C03648=1197.053,12.345,-44.404,-179.678,5.675,148.906
C03649=1197.057,12.095,-44.389,-179.681,5.675,148.907
C03650=1197.063,11.846,-44.375,-179.684,5.674,148.908
C03651=1197.069,11.596,-44.360,-179.686,5.674,148.908
C03652=1197.074,11.347,-44.346,-179.689,5.673,148.909
C03653=1197.079,11.097,-44.331,-179.691,5.672,148.910
C03654=1197.084,10.847,-44.317,-179.694,5.672,148.910
C03655=1197.088,10.598,-44.302,-179.697,5.671,148.911
C03656=1197.093,10.349,-44.288,-179.699,5.671,148.912
C03657=1197.099,10.100,-44.274,-179.702,5.670,148.912
C03658=1197.104,9.850,-44.260,-179.704,5.669,148.913
C03659=1197.109,9.600,-44.245,-179.707,5.669,148.914
C03660=1197.114,9.350,-44.231,-179.709,5.669,148.914
C03661=1197.119,9.101,-44.217,-179.712,5.668,148.915
C03662=1197.123,8.851,-44.203,-179.714,5.667,148.915
C03663=1197.129,8.602,-44.189,-179.717,5.667,148.916
C03664=1197.134,8.352,-44.174,-179.719,5.667,148.917
C03665=1197.139,8.103,-44.159,-179.721,5.666,148.917
C03666=1197.144,7.853,-44.145,-179.724,5.666,148.918
C03667=1197.149,7.604,-44.131,-179.726,5.665,148.919
C03668=1197.154,7.355,-44.117,-179.729,5.665,148.919
C03669=1197.159,7.105,-44.103,-179.732,5.664,148.920
C03670=1197.164,6.855,-44.088,-179.734,5.664,148.921
C03671=1197.169,6.606,-44.074,-179.737,5.663,148.921
C03672=1197.174,6.356,-44.060,-179.739,5.662,148.922
C03673=1197.179,6.107,-44.046,-179.742,5.662,148.922
C03674=1197.184,5.857,-44.032,-179.744,5.661,148.923
C03675=1197.189,5.607,-44.017,-179.747,5.661,148.924
C03676=1197.194,5.358,-44.003,-179.750,5.660,148.924
C03677=1197.200,5.109,-43.989,-179.751,5.660,148.925
C03678=1197.205,4.858,-43.976,-179.754,5.660,148.926
C03679=1197.209,4.609,-43.962,-179.757,5.659,148.926
C03680=1197.214,4.359,-43.948,-179.759,5.659,148.927
C03681=1197.220,4.110,-43.934,-179.762,5.658,148.928
C03682=1197.225,3.861,-43.919,-179.764,5.657,148.928
C03683=1197.230,3.611,-43.905,-179.767,5.657,148.929
C03684=1197.235,3.361,-43.891,-179.769,5.656,148.930
C03685=1197.241,3.092,-43.876,-179.772,5.656,148.930
C03686=1197.246,2.824,-43.861,-179.775,5.655,148.931
C03687=1197.251,2.554,-43.846,-179.777,5.655,148.932
C03688=1197.257,2.285,-43.831,-179.780,5.654,148.932
C03689=1197.262,2.035,-43.816,-179.783,5.654,148.933
C03690=1197.267,1.786,-43.802,-179.785,5.653,148.934
C03691=1197.272,1.536,-43.788,-179.788,5.653,148.934
C03692=1197.277,1.286,-43.775,-179.790,5.652,148.935
C03693=1197.282,1.037,-43.761,-179.793,5.652,148.935
C03694=1197.287,0.788,-43.747,-179.795,5.652,148.936
C03695=1197.292,0.538,-43.733,-179.797,5.651,148.937
C03696=1197.298,0.289,-43.719,-179.800,5.651,148.938
C03697=1197.303,0.039,-43.705,-179.802,5.650,148.938
C03698=1197.307,-0.211,-43.692,-179.805,5.650,148.939
C03699=1197.313,-0.460,-43.678,-179.808,5.649,148.939
C03700=1197.318,-0.710,-43.663,-179.810,5.649,148.940
C03701=1197.323,-0.959,-43.649,-179.813,5.648,148.941
C03702=1197.329,-1.209,-43.636,-179.815,5.647,148.941
C03703=1197.333,-1.458,-43.622,-179.817,5.648,148.942
C03704=1197.338,-1.708,-43.608,-179.820,5.647,148.943
C03705=1197.343,-1.957,-43.594,-179.822,5.647,148.943
C03706=1197.349,-2.207,-43.580,-179.825,5.646,148.944
C03707=1197.353,-2.457,-43.567,-179.827,5.645,148.944
C03708=1197.358,-2.706,-43.553,-179.830,5.645,148.945
C03709=1197.364,-2.956,-43.539,-179.833,5.644,148.946
C03710=1197.369,-3.206,-43.525,-179.835,5.644,148.947
C03711=1197.373,-3.454,-43.512,-179.837,5.644,148.947
C03712=1197.379,-3.705,-43.498,-179.840,5.644,148.948
C03713=1197.384,-3.954,-43.484,-179.842,5.643,148.948
C03714=1197.389,-4.204,-43.470,-179.845,5.642,148.949
C03715=1197.394,-4.454,-43.457,-179.847,5.642,148.950
C03716=1197.399,-4.703,-43.443,-179.850,5.641,148.950
C03717=1197.404,-4.952,-43.429,-179.853,5.641,148.951
C03718=1197.409,-5.203,-43.415,-179.855,5.640,148.952
C03719=1197.414,-5.451,-43.402,-179.857,5.640,148.952
C03720=1197.419,-5.701,-43.388,-179.860,5.640,148.953
C03721=1197.425,-5.951,-43.374,-179.862,5.639,148.954
C03722=1197.429,-6.200,-43.361,-179.865,5.639,148.954
C03723=1197.435,-6.450,-43.347,-179.867,5.638,148.955
C03724=1197.440,-6.699,-43.333,-179.870,5.638,148.955
C03725=1197.445,-6.949,-43.320,-179.872,5.637,148.956
C03726=1197.450,-7.198,-43.306,-179.874,5.637,148.957
C03727=1197.455,-7.448,-43.292,-179.877,5.637,148.958
C03728=1197.460,-7.698,-43.279,-179.880,5.636,148.958
C03729=1197.465,-7.947,-43.265,-179.882,5.636,148.959
C03730=1197.470,-8.197,-43.252,-179.885,5.635,148.959
C03731=1197.475,-8.446,-43.238,-179.887,5.635,148.960
C03732=1197.481,-8.696,-43.225,-179.890,5.634,148.961
C03733=1197.485,-8.945,-43.211,-179.892,5.634,148.961
C03734=1197.491,-9.196,-43.198,-179.894,5.634,148.962
C03735=1197.495,-9.444,-43.185,-179.897,5.633,148.963
C03736=1197.501,-9.695,-43.171,-179.899,5.633,148.963
C03737=1197.506,-9.944,-43.157,-179.902,5.632,148.964
C03738=1197.511,-10.194,-43.144,-179.905,5.632,148.965
C03739=1197.516,-10.443,-43.130,-179.907,5.631,148.965
C03740=1197.521,-10.693,-43.117,-179.909,5.631,148.966
C03741=1197.526,-10.942,-43.103,-179.912,5.631,148.967
C03742=1197.532,-11.192,-43.090,-179.914,5.630,148.967
C03743=1197.536,-11.442,-43.077,-179.917,5.630,148.968
C03744=1197.542,-11.691,-43.063,-179.920,5.629,148.969
C03745=1197.546,-11.941,-43.050,-179.922,5.628,148.969
C03746=1197.552,-12.190,-43.036,-179.924,5.629,148.970
C03747=1197.556,-12.440,-43.023,-179.927,5.628,148.970
C03748=1197.562,-12.690,-43.010,-179.929,5.628,148.971
C03749=1197.566,-12.939,-42.996,-179.932,5.627,148.972
C03750=1197.572,-13.189,-42.983,-179.934,5.626,148.972
C03751=1197.577,-13.438,-42.969,-179.937,5.626,148.973
C03752=1197.582,-13.688,-42.956,-179.939,5.626,148.974
C03753=1197.587,-13.938,-42.943,-179.941,5.626,148.974
C03754=1197.592,-14.187,-42.929,-179.944,5.625,148.975
C03755=1197.597,-14.437,-42.916,-179.947,5.625,148.976
C03756=1197.603,-14.686,-42.903,-179.949,5.624,148.976
C03757=1197.608,-14.935,-42.890,-179.952,5.623,148.977
C03758=1197.613,-15.185,-42.876,-179.954,5.624,148.978
C03759=1197.618,-15.435,-42.864,-179.956,5.623,148.978
C03760=1197.623,-15.685,-42.850,-179.959,5.623,148.979
C03761=1197.628,-15.934,-42.837,-179.961,5.622,148.980
C03762=1197.633,-16.184,-42.823,-179.964,5.622,148.980
C03763=1197.639,-16.433,-42.811,-179.966,5.622,148.981
C03764=1197.643,-16.683,-42.797,-179.969,5.621,148.982
C03765=1197.649,-16.932,-42.784,-179.971,5.621,148.982
C03766=1197.654,-17.182,-42.771,-179.974,5.620,148.983
C03767=1197.659,-17.432,-42.758,-179.976,5.620,148.983
C03768=1197.664,-17.681,-42.744,-179.979,5.619,148.984
C03769=1197.669,-17.931,-42.731,-179.981,5.619,148.985
C03770=1197.674,-18.180,-42.718,-179.983,5.619,148.986
C03771=1197.679,-18.430,-42.705,-179.986,5.619,148.986
C03772=1197.685,-18.680,-42.692,-179.989,5.618,148.987
C03773=1197.689,-18.929,-42.679,-179.991,5.617,148.987
C03774=1197.695,-19.179,-42.665,-179.993,5.618,148.988
C03775=1197.700,-19.428,-42.652,-179.996,5.617,148.989
C03776=1197.704,-19.678,-42.639,-179.998,5.617,148.989
C03777=1197.710,-19.928,-42.626,179.999,5.616,148.990
C03778=1197.715,-20.177,-42.614,179.997,5.615,148.991
C03779=1197.720,-20.427,-42.599,179.995,5.616,148.991
C03780=1197.725,-20.676,-42.587,179.992,5.615,148.992
C03781=1197.730,-20.926,-42.574,179.989,5.615,148.993
C03782=1197.736,-21.176,-42.561,179.987,5.614,148.993
C03783=1197.741,-21.425,-42.548,179.984,5.614,148.994
C03784=1197.746,-21.675,-42.535,179.983,5.614,148.995
C03785=1197.751,-21.925,-42.522,179.980,5.613,148.995
C03786=1197.756,-22.174,-42.509,179.977,5.613,148.996
C03787=1197.761,-22.424,-42.496,179.975,5.612,148.997
C03788=1197.766,-22.673,-42.482,179.972,5.612,148.997
C03789=1197.771,-22.943,-42.469,179.969,5.611,148.998
C03790=1197.778,-23.212,-42.455,179.967,5.612,148.999
C03791=1197.783,-23.482,-42.441,179.965,5.611,148.999
C03792=1197.789,-23.752,-42.427,179.962,5.611,149.000
C03793=1197.794,-24.001,-42.414,179.959,5.610,149.001
C03794=1197.799,-24.251,-42.402,179.957,5.610,149.002
C03795=1197.803,-24.501,-42.389,179.954,5.609,149.002
C03796=1197.809,-24.750,-42.375,179.952,5.609,149.003
C03797=1197.814,-25.000,-42.363,179.950,5.609,149.003
C03798=1197.819,-25.250,-42.350,179.947,5.608,149.004
C03799=1197.824,-25.499,-42.337,179.944,5.608,149.005
C03800=1197.830,-25.749,-42.324,179.942,5.607,149.005
C03801=1197.835,-25.998,-42.312,179.940,5.607,149.006
C03802=1197.839,-26.248,-42.299,179.937,5.607,149.007
C03803=1197.845,-26.497,-42.286,179.935,5.606,149.007
C03804=1197.850,-26.747,-42.273,179.932,5.606,149.008
C03805=1197.855,-26.997,-42.260,179.930,5.606,149.009
C03806=1197.860,-27.246,-42.247,179.928,5.605,149.009
C03807=1197.865,-27.496,-42.235,179.925,5.605,149.010
C03808=1197.870,-27.746,-42.222,179.923,5.605,149.011
C03809=1197.876,-27.995,-42.208,179.920,5.604,149.011
C03810=1197.881,-28.245,-42.196,179.918,5.604,149.012
C03811=1197.886,-28.495,-42.184,179.915,5.604,149.013
C03812=1197.891,-28.745,-42.171,179.913,5.603,149.013
C03813=1197.896,-28.994,-42.158,179.910,5.603,149.014
C03814=1197.901,-29.243,-42.146,179.908,5.603,149.015
C03815=1197.907,-29.493,-42.133,179.906,5.602,149.015
C03816=1197.911,-29.743,-42.120,179.903,5.602,149.016
C03817=1197.916,-29.992,-42.107,179.901,5.601,149.016
C03818=1197.922,-30.242,-42.094,179.899,5.602,149.017
C03819=1197.927,-30.491,-42.083,179.896,5.601,149.018
C03820=1197.931,-30.741,-42.070,179.893,5.601,149.019
C03821=1197.937,-30.991,-42.057,179.891,5.600,149.019
C03822=1197.942,-31.240,-42.044,179.889,5.600,149.020
C03823=1197.948,-31.490,-42.031,179.886,5.600,149.020
C03824=1197.953,-31.740,-42.019,179.884,5.599,149.021
C03825=1197.958,-31.990,-42.006,179.881,5.599,149.022
C03826=1197.963,-32.239,-41.994,179.879,5.599,149.022
C03827=1197.968,-32.488,-41.981,179.876,5.599,149.023
C03828=1197.973,-32.738,-41.968,179.874,5.598,149.024
C03829=1197.978,-32.988,-41.957,179.872,5.597,149.024
C03830=1197.983,-33.238,-41.944,179.869,5.598,149.025
C03831=1197.988,-33.487,-41.931,179.867,5.597,149.026
C03832=1197.994,-33.737,-41.918,179.864,5.597,149.026
C03833=1197.999,-33.986,-41.906,179.861,5.596,149.027
C03834=1198.004,-34.236,-41.893,179.860,5.596,149.028
C03835=1198.009,-34.486,-41.880,179.857,5.596,149.028
C03836=1198.014,-34.736,-41.869,179.855,5.595,149.029
C03837=1198.019,-34.985,-41.856,179.852,5.595,149.030
C03838=1198.025,-35.234,-41.843,179.850,5.595,149.030
C03839=1198.030,-35.484,-41.831,179.847,5.595,149.031
C03840=1198.035,-35.734,-41.819,179.845,5.594,149.032
C03841=1198.040,-35.984,-41.806,179.842,5.593,149.032
C03842=1198.045,-36.233,-41.793,179.840,5.594,149.033
C03843=1198.050,-36.483,-41.781,179.838,5.593,149.034
C03844=1198.055,-36.732,-41.769,179.835,5.593,149.034
C03845=1198.061,-36.982,-41.757,179.833,5.592,149.035
C03846=1198.066,-37.231,-41.744,179.831,5.592,149.036
C03847=1198.071,-37.481,-41.732,179.828,5.592,149.036
C03848=1198.076,-37.731,-41.720,179.825,5.591,149.037
C03849=1198.081,-37.981,-41.707,179.823,5.591,149.038
C03850=1198.086,-38.230,-41.694,179.821,5.591,149.038
C03851=1198.092,-38.480,-41.682,179.818,5.590,149.039
C03852=1198.097,-38.729,-41.670,179.816,5.590,149.040
C03853=1198.102,-38.979,-41.658,179.814,5.590,149.040
C03854=1198.107,-39.229,-41.645,179.811,5.590,149.041
C03855=1198.113,-39.479,-41.633,179.808,5.589,149.042
C03856=1198.118,-39.728,-41.621,179.806,5.589,149.042
C03857=1198.123,-39.977,-41.608,179.804,5.589,149.043
C03858=1198.128,-40.228,-41.596,179.801,5.589,149.043
C03859=1198.132,-40.477,-41.584,179.799,5.588,149.044
C03860=1198.138,-40.727,-41.572,179.797,5.588,149.045
C03861=1198.143,-40.976,-41.559,179.794,5.588,149.046
C03862=1198.148,-41.226,-41.548,179.792,5.587,149.046
C03863=1198.153,-41.475,-41.535,179.789,5.587,149.047
C03864=1198.159,-41.725,-41.523,179.787,5.587,149.047
C03865=1198.164,-41.975,-41.510,179.784,5.587,149.048
C03866=1198.169,-42.224,-41.499,179.782,5.586,149.049
C03867=1198.174,-42.474,-41.486,179.780,5.586,149.049
C03868=1198.180,-42.724,-41.474,179.777,5.586,149.050
C03869=1198.184,-42.973,-41.462,179.775,5.585,149.051
C03870=1198.190,-43.223,-41.450,179.772,5.585,149.051
C03871=1198.195,-43.473,-41.438,179.770,5.585,149.052
C03872=1198.200,-43.723,-41.425,179.767,5.585,149.053
C03873=1198.205,-43.973,-41.413,179.765,5.584,149.053
C03874=1198.210,-44.222,-41.401,179.763,5.584,149.054
C03875=1198.215,-44.472,-41.390,179.760,5.584,149.055
C03876=1198.220,-44.721,-41.377,179.758,5.583,149.055
C03877=1198.225,-44.971,-41.365,179.755,5.583,149.056
C03878=1198.231,-45.221,-41.353,179.754,5.583,149.057
C03879=1198.236,-45.470,-41.341,179.751,5.582,149.057
C03880=1198.241,-45.720,-41.329,179.748,5.582,149.058
C03881=1198.246,-45.969,-41.317,179.746,5.582,149.059
C03882=1198.251,-46.219,-41.305,179.743,5.582,149.059
C03883=1198.257,-46.469,-41.293,179.741,5.581,149.060
C03884=1198.262,-46.718,-41.280,179.739,5.581,149.061
C03885=1198.267,-46.968,-41.268,179.737,5.581,149.061
C03886=1198.272,-47.218,-41.257,179.734,5.580,149.062
C03887=1198.277,-47.467,-41.245,179.731,5.580,149.063
C03888=1198.282,-47.717,-41.233,179.729,5.580,149.063
C03889=1198.288,-47.967,-41.221,179.727,5.579,149.064
C03890=1198.292,-48.216,-41.209,179.724,5.579,149.065
C03891=1198.298,-48.466,-41.197,179.722,5.579,149.065
C03892=1198.303,-48.716,-41.185,179.720,5.579,149.066
C03893=1198.309,-48.985,-41.172,179.717,5.578,149.067
C03894=1198.314,-49.256,-41.159,179.714,5.578,149.067
C03895=1198.320,-49.526,-41.146,179.712,5.578,149.068
C03896=1198.325,-49.796,-41.134,179.709,5.578,149.069
C03897=1198.331,-50.046,-41.122,179.707,5.577,149.069
C03898=1198.336,-50.295,-41.109,179.704,5.577,149.070
C03899=1198.341,-50.545,-41.098,179.703,5.577,149.071
C03900=1198.346,-50.795,-41.086,179.700,5.577,149.071
C03901=1198.352,-51.045,-41.074,179.697,5.576,149.072
C03902=1198.357,-51.295,-41.062,179.695,5.576,149.073
C03903=1198.361,-51.544,-41.050,179.692,5.576,149.073
C03904=1198.367,-51.793,-41.039,179.690,5.576,149.074
C03905=1198.372,-52.043,-41.027,179.688,5.576,149.075
C03906=1198.377,-52.293,-41.015,179.686,5.575,149.075
C03907=1198.382,-52.543,-41.003,179.683,5.575,149.076
C03908=1198.388,-52.792,-40.991,179.681,5.575,149.077
C03909=1198.393,-53.041,-40.980,179.678,5.575,149.077
C03910=1198.398,-53.291,-40.968,179.676,5.574,149.078
C03911=1198.404,-53.541,-40.956,179.674,5.574,149.079
C03912=1198.408,-53.791,-40.945,179.671,5.574,149.079
C03913=1198.414,-54.041,-40.933,179.669,5.573,149.080
C03914=1198.418,-54.290,-40.921,179.666,5.574,149.081
C03915=1198.424,-54.540,-40.909,179.664,5.573,149.081
C03916=1198.429,-54.790,-40.897,179.662,5.572,149.082
C03917=1198.434,-55.039,-40.886,179.660,5.573,149.083
C03918=1198.439,-55.289,-40.874,179.657,5.572,149.083
C03919=1198.444,-55.538,-40.863,179.654,5.572,149.084
C03920=1198.450,-55.788,-40.851,179.653,5.572,149.085
C03921=1198.455,-56.038,-40.839,179.650,5.571,149.085
C03922=1198.460,-56.287,-40.828,179.647,5.571,149.086
C03923=1198.465,-56.537,-40.816,179.645,5.571,149.087
C03924=1198.470,-56.787,-40.805,179.643,5.571,149.087
C03925=1198.476,-57.037,-40.793,179.640,5.570,149.088
C03926=1198.482,-57.286,-40.782,179.638,5.570,149.089
C03927=1198.486,-57.535,-40.770,179.636,5.570,149.089
C03928=1198.491,-57.785,-40.758,179.633,5.569,149.090
C03929=1198.496,-58.035,-40.746,179.631,5.570,149.091
C03930=1198.501,-58.285,-40.734,179.629,5.569,149.091
C03931=1198.506,-58.534,-40.723,179.626,5.569,149.092
C03932=1198.512,-58.784,-40.711,179.624,5.569,149.093
C03933=1198.517,-59.033,-40.700,179.621,5.568,149.093
C03934=1198.522,-59.283,-40.688,179.619,5.568,149.094
C03935=1198.527,-59.533,-40.677,179.617,5.568,149.094
C03936=1198.532,-59.783,-40.665,179.614,5.568,149.095
C03937=1198.537,-60.033,-40.655,179.612,5.567,149.096
C03938=1198.543,-60.283,-40.643,179.610,5.567,149.097
C03939=1198.548,-60.532,-40.632,179.607,5.567,149.097
C03940=1198.554,-60.782,-40.620,179.605,5.567,149.098
C03941=1198.558,-61.031,-40.609,179.603,5.567,149.098
C03942=1198.564,-61.281,-40.597,179.600,5.566,149.099
C03943=1198.568,-61.531,-40.586,179.598,5.566,149.100
C03944=1198.574,-61.780,-40.574,179.595,5.566,149.101
C03945=1198.579,-62.030,-40.563,179.593,5.565,149.101
C03946=1198.585,-62.280,-40.551,179.591,5.566,149.102
C03947=1198.589,-62.529,-40.540,179.588,5.565,149.102
C03948=1198.595,-62.779,-40.528,179.586,5.565,149.103
C03949=1198.600,-63.029,-40.517,179.584,5.565,149.104
C03950=1198.606,-63.279,-40.506,179.581,5.564,149.104
C03951=1198.610,-63.528,-40.494,179.579,5.564,149.105
C03952=1198.615,-63.778,-40.483,179.577,5.564,149.106
C03953=1198.621,-64.027,-40.471,179.574,5.564,149.106
C03954=1198.626,-64.277,-40.460,179.572,5.564,149.107
C03955=1198.631,-64.527,-40.448,179.570,5.563,149.108
C03956=1198.636,-64.777,-40.438,179.567,5.563,149.108
C03957=1198.642,-65.026,-40.427,179.565,5.563,149.109
C03958=1198.647,-65.276,-40.415,179.562,5.563,149.110
C03959=1198.652,-65.526,-40.404,179.560,5.562,149.110
C03960=1198.657,-65.776,-40.392,179.558,5.562,149.111
C03961=1198.663,-66.025,-40.382,179.555,5.562,149.112
C03962=1198.667,-66.275,-40.370,179.553,5.562,149.112
C03963=1198.673,-66.525,-40.358,179.551,5.562,149.113
C03964=1198.678,-66.774,-40.347,179.548,5.561,149.113
C03965=1198.684,-67.024,-40.336,179.546,5.561,149.114
C03966=1198.689,-67.274,-40.325,179.544,5.561,149.115
C03967=1198.693,-67.523,-40.314,179.541,5.560,149.116
C03968=1198.699,-67.773,-40.302,179.539,5.561,149.116
C03969=1198.704,-68.023,-40.292,179.537,5.560,149.117
C03970=1198.709,-68.272,-40.280,179.535,5.560,149.117
C03971=1198.715,-68.522,-40.269,179.532,5.560,149.118
C03972=1198.720,-68.771,-40.258,179.529,5.560,149.119
C03973=1198.725,-69.022,-40.247,179.527,5.560,149.120
C03974=1198.730,-69.271,-40.235,179.525,5.559,149.120
C03975=1198.735,-69.520,-40.224,179.522,5.559,149.121
C03976=1198.740,-69.771,-40.214,179.520,5.559,149.122
C03977=1198.746,-70.021,-40.202,179.518,5.559,149.122
C03978=1198.751,-70.270,-40.191,179.516,5.559,149.123
C03979=1198.756,-70.520,-40.180,179.513,5.558,149.123
C03980=1198.762,-70.770,-40.168,179.511,5.558,149.124
C03981=1198.767,-71.019,-40.157,179.509,5.558,149.125
C03982=1198.772,-71.269,-40.147,179.506,5.558,149.126
C03983=1198.777,-71.518,-40.135,179.504,5.558,149.126
C03984=1198.783,-71.768,-40.124,179.502,5.557,149.127
C03985=1198.788,-72.018,-40.113,179.499,5.557,149.127
C03986=1198.793,-72.267,-40.102,179.497,5.557,149.128
C03987=1198.799,-72.517,-40.091,179.495,5.556,149.129
C03988=1198.803,-72.767,-40.080,179.493,5.557,149.129
C03989=1198.809,-73.016,-40.069,179.490,5.556,149.130
C03990=1198.814,-73.266,-40.059,179.487,5.556,149.131
C03991=1198.819,-73.516,-40.047,179.486,5.556,149.131
C03992=1198.825,-73.766,-40.036,179.483,5.555,149.132
C03993=1198.829,-74.015,-40.025,179.481,5.556,149.133
C03994=1198.835,-74.265,-40.015,179.478,5.555,149.133
C03995=1198.840,-74.515,-40.004,179.476,5.555,149.134
C03996=1198.845,-74.765,-39.992,179.474,5.555,149.135
C03997=1198.851,-75.035,-39.981,179.471,5.554,149.135
C03998=1198.856,-75.306,-39.969,179.469,5.554,149.136
C03999=1198.862,-75.577,-39.957,179.467,5.554,149.137
C04000=1198.868,-75.847,-39.945,179.464,5.554,149.137
C04001=1198.873,-76.098,-39.934,179.461,5.554,149.138
C04002=1198.879,-76.346,-39.923,179.459,5.554,149.139
C04003=1198.884,-76.597,-39.913,179.456,5.554,149.139
C04004=1198.888,-76.846,-39.901,179.454,5.553,149.140
C04005=1198.894,-77.096,-39.891,179.452,5.553,149.141
C04006=1198.899,-77.346,-39.879,179.449,5.553,149.141
C04007=1198.905,-77.595,-39.869,179.447,5.553,149.142
C04008=1198.910,-77.845,-39.858,179.445,5.552,149.143
C04009=1198.915,-78.095,-39.848,179.443,5.552,149.143
C04010=1198.920,-78.345,-39.837,179.440,5.552,149.144
C04011=1198.925,-78.594,-39.826,179.438,5.552,149.145
C04012=1198.931,-78.844,-39.815,179.436,5.552,149.145
C04013=1198.936,-79.094,-39.804,179.434,5.551,149.146
C04014=1198.941,-79.343,-39.793,179.431,5.552,149.147
C04015=1198.946,-79.593,-39.782,179.429,5.551,149.147
C04016=1198.952,-79.843,-39.772,179.426,5.551,149.148
C04017=1198.957,-80.093,-39.761,179.425,5.551,149.148
C04018=1198.962,-80.342,-39.750,179.422,5.550,149.149
C04019=1198.967,-80.592,-39.740,179.420,5.551,149.150
C04020=1198.973,-80.842,-39.730,179.417,5.550,149.151
C04021=1198.977,-81.091,-39.718,179.415,5.550,149.151
C04022=1198.983,-81.342,-39.707,179.413,5.550,149.152
C04023=1198.988,-81.591,-39.696,179.410,5.549,149.153
C04024=1198.993,-81.841,-39.686,179.408,5.550,149.153
C04025=1198.999,-82.090,-39.676,179.406,5.549,149.154
C04026=1199.004,-82.340,-39.664,179.404,5.549,149.154
C04027=1199.009,-82.590,-39.654,179.401,5.549,149.155
C04028=1199.014,-82.840,-39.643,179.398,5.549,149.156
C04029=1199.020,-83.089,-39.633,179.397,5.549,149.156
C04030=1199.025,-83.339,-39.622,179.394,5.548,149.157
C04031=1199.030,-83.589,-39.612,179.392,5.549,149.158
C04032=1199.035,-83.839,-39.601,179.389,5.548,149.158
C04033=1199.040,-84.088,-39.590,179.388,5.548,149.159
C04034=1199.045,-84.338,-39.580,179.385,5.548,149.160
C04035=1199.051,-84.588,-39.569,179.382,5.547,149.160
C04036=1199.056,-84.838,-39.559,179.380,5.548,149.161
C04037=1199.061,-85.087,-39.548,179.378,5.547,149.162
C04038=1199.066,-85.337,-39.537,179.376,5.547,149.162
C04039=1199.072,-85.586,-39.527,179.373,5.547,149.163
C04040=1199.077,-85.836,-39.517,179.371,5.547,149.164
C04041=1199.082,-86.086,-39.506,179.369,5.546,149.164
C04042=1199.088,-86.335,-39.495,179.366,5.546,149.165
C04043=1199.093,-86.585,-39.485,179.364,5.546,149.166
C04044=1199.098,-86.835,-39.475,179.362,5.546,149.166
C04045=1199.103,-87.085,-39.463,179.360,5.546,149.167
C04046=1199.109,-87.334,-39.453,179.357,5.545,149.167
C04047=1199.114,-87.584,-39.443,179.355,5.546,149.168
C04048=1199.119,-87.834,-39.432,179.353,5.545,149.169
C04049=1199.124,-88.084,-39.422,179.351,5.545,149.169
C04050=1199.130,-88.334,-39.412,179.348,5.545,149.170
C04051=1199.135,-88.583,-39.401,179.346,5.545,149.171
C04052=1199.139,-88.833,-39.391,179.344,5.545,149.171
C04053=1199.145,-89.082,-39.380,179.341,5.544,149.172
C04054=1199.150,-89.332,-39.370,179.339,5.545,149.173
C04055=1199.156,-89.582,-39.360,179.337,5.544,149.173
C04056=1199.161,-89.832,-39.349,179.335,5.544,149.174
C04057=1199.166,-90.082,-39.339,179.332,5.544,149.175
C04058=1199.172,-90.331,-39.329,179.330,5.544,149.175
C04059=1199.176,-90.581,-39.317,179.328,5.544,149.176
C04060=1199.182,-90.830,-39.307,179.326,5.543,149.177
C04061=1199.187,-91.081,-39.297,179.323,5.543,149.177
C04062=1199.192,-91.330,-39.287,179.321,5.543,149.178
C04063=1199.198,-91.579,-39.277,179.319,5.543,149.178
C04064=1199.203,-91.830,-39.266,179.316,5.542,149.179
C04065=1199.208,-92.079,-39.256,179.314,5.543,149.180
C04066=1199.214,-92.329,-39.246,179.312,5.542,149.181
C04067=1199.219,-92.579,-39.235,179.310,5.542,149.181
C04068=1199.224,-92.829,-39.225,179.307,5.542,149.182
C04069=1199.229,-93.078,-39.215,179.305,5.542,149.182
C04070=1199.234,-93.328,-39.205,179.303,5.542,149.183
C04071=1199.240,-93.578,-39.195,179.301,5.541,149.184
C04072=1199.245,-93.828,-39.184,179.298,5.542,149.184
C04073=1199.250,-94.077,-39.174,179.296,5.541,149.185
C04074=1199.256,-94.327,-39.164,179.294,5.541,149.186
C04075=1199.260,-94.577,-39.154,179.291,5.541,149.186
C04076=1199.266,-94.826,-39.143,179.289,5.541,149.187
C04077=1199.271,-95.076,-39.133,179.287,5.541,149.188
C04078=1199.276,-95.326,-39.123,179.285,5.541,149.188
C04079=1199.282,-95.576,-39.112,179.282,5.540,149.189
C04080=1199.287,-95.825,-39.103,179.280,5.541,149.190
C04081=1199.292,-96.075,-39.092,179.278,5.540,149.190
C04082=1199.297,-96.325,-39.082,179.275,5.539,149.191
C04083=1199.303,-96.574,-39.072,179.273,5.540,149.192
C04084=1199.308,-96.825,-39.061,179.271,5.539,149.192
C04085=1199.313,-97.074,-39.052,179.269,5.539,149.193
C04086=1199.319,-97.323,-39.041,179.266,5.539,149.193
C04087=1199.324,-97.574,-39.031,179.264,5.539,149.194
C04088=1199.329,-97.823,-39.021,179.262,5.539,149.195
C04089=1199.334,-98.073,-39.012,179.260,5.539,149.195
C04090=1199.340,-98.322,-39.002,179.257,5.539,149.196
C04091=1199.345,-98.573,-38.991,179.256,5.539,149.197
C04092=1199.350,-98.822,-38.981,179.253,5.538,149.197
C04093=1199.355,-99.071,-38.971,179.251,5.539,149.198
C04094=1199.360,-99.322,-38.961,179.248,5.538,149.199
C04095=1199.366,-99.571,-38.950,179.247,5.538,149.199
C04096=1199.372,-99.821,-38.940,179.244,5.538,149.200
C04097=1199.377,-100.071,-38.931,179.242,5.538,149.201
C04098=1199.382,-100.321,-38.921,179.240,5.537,149.201
C04099=1199.387,-100.570,-38.911,179.237,5.537,149.202
C04100=1199.392,-100.820,-38.901,179.235,5.537,149.202
C04101=1199.398,-101.091,-38.889,179.232,5.537,149.203
C04102=1199.404,-101.363,-38.879,179.230,5.537,149.204
C04103=1199.409,-101.635,-38.868,179.228,5.536,149.204
C04104=1199.415,-101.905,-38.857,179.225,5.536,149.205
C04105=1199.420,-102.155,-38.848,179.223,5.536,149.206
C04106=1199.425,-102.406,-38.838,179.221,5.536,149.207
C04107=1199.431,-102.655,-38.827,179.219,5.536,149.207
C04108=1199.436,-102.904,-38.818,179.216,5.536,149.208
C04109=1199.442,-103.154,-38.808,179.214,5.536,149.208
C04110=1199.447,-103.405,-38.798,179.212,5.536,149.209
C04111=1199.452,-103.654,-38.788,179.210,5.536,149.210
C04112=1199.457,-103.903,-38.778,179.207,5.535,149.210
C04113=1199.463,-104.154,-38.768,179.205,5.536,149.211
C04114=1199.467,-104.404,-38.758,179.203,5.535,149.212
C04115=1199.473,-104.653,-38.748,179.201,5.535,149.212
C04116=1199.478,-104.902,-38.739,179.198,5.535,149.213
C04117=1199.484,-105.153,-38.729,179.197,5.535,149.213
C04118=1199.489,-105.402,-38.719,179.194,5.534,149.214
C04119=1199.494,-105.652,-38.709,179.192,5.535,149.215
C04120=1199.500,-105.902,-38.699,179.190,5.534,149.215
C04121=1199.504,-106.151,-38.690,179.188,5.534,149.216
C04122=1199.510,-106.401,-38.680,179.185,5.534,149.217
C04123=1199.516,-106.651,-38.670,179.183,5.534,149.217
C04124=1199.520,-106.901,-38.660,179.181,5.534,149.218
C04125=1199.526,-107.151,-38.650,179.179,5.534,149.219
C04126=1199.531,-107.400,-38.641,179.176,5.533,149.219
C04127=1199.537,-107.650,-38.631,179.174,5.534,149.220
C04128=1199.541,-107.899,-38.621,179.172,5.533,149.221
C04129=1199.547,-108.150,-38.611,179.170,5.533,149.221
C04130=1199.552,-108.400,-38.601,179.167,5.533,149.222
C04131=1199.557,-108.649,-38.591,179.165,5.533,149.223
C04132=1199.563,-108.899,-38.582,179.163,5.532,149.223
C04133=1199.568,-109.148,-38.572,179.161,5.533,149.224
C04134=1199.574,-109.398,-38.563,179.158,5.532,149.224
C04135=1199.578,-109.648,-38.553,179.157,5.532,149.225
C04136=1199.584,-109.898,-38.543,179.154,5.532,149.226
C04137=1199.589,-110.148,-38.534,179.152,5.532,149.226
C04138=1199.594,-110.397,-38.524,179.150,5.532,149.227
C04139=1199.600,-110.647,-38.515,179.148,5.532,149.228
C04140=1199.605,-110.897,-38.504,179.145,5.532,149.228
C04141=1199.610,-111.146,-38.496,179.143,5.532,149.229
C04142=1199.616,-111.396,-38.485,179.141,5.531,149.229
C04143=1199.621,-111.647,-38.476,179.139,5.532,149.230
C04144=1199.626,-111.896,-38.466,179.136,5.531,149.231
C04145=1199.631,-112.146,-38.457,179.134,5.531,149.231
C04146=1199.637,-112.396,-38.447,179.132,5.531,149.232
C04147=1199.642,-112.645,-38.437,179.130,5.531,149.233
C04148=1199.648,-112.895,-38.428,179.127,5.530,149.233
C04149=1199.653,-113.144,-38.418,179.125,5.531,149.234
C04150=1199.658,-113.394,-38.409,179.123,5.530,149.235
C04151=1199.664,-113.644,-38.400,179.121,5.530,149.235
C04152=1199.668,-113.894,-38.390,179.118,5.530,149.236
C04153=1199.674,-114.144,-38.380,179.117,5.530,149.236
C04154=1199.679,-114.394,-38.371,179.114,5.530,149.237
C04155=1199.685,-114.644,-38.361,179.113,5.530,149.238
C04156=1199.689,-114.893,-38.351,179.110,5.529,149.238
C04157=1199.695,-115.143,-38.342,179.108,5.530,149.239
C04158=1199.700,-115.392,-38.332,179.106,5.529,149.240
C04159=1199.705,-115.642,-38.323,179.103,5.529,149.240
C04160=1199.711,-115.892,-38.313,179.101,5.529,149.241
C04161=1199.716,-116.142,-38.304,179.099,5.529,149.241
C04162=1199.722,-116.392,-38.295,179.097,5.528,149.242
C04163=1199.727,-116.641,-38.285,179.094,5.529,149.243
C04164=1199.732,-116.891,-38.276,179.092,5.528,149.243
C04165=1199.738,-117.140,-38.266,179.090,5.528,149.244
C04166=1199.742,-117.391,-38.257,179.088,5.528,149.245
C04167=1199.748,-117.641,-38.247,179.086,5.528,149.245
C04168=1199.753,-117.890,-38.238,179.083,5.528,149.246
C04169=1199.758,-118.140,-38.229,179.082,5.528,149.246
C04170=1199.764,-118.390,-38.219,179.079,5.527,149.247
C04171=1199.769,-118.640,-38.210,179.077,5.528,149.248
C04172=1199.774,-118.889,-38.201,179.075,5.527,149.248
C04173=1199.780,-119.140,-38.191,179.073,5.527,149.249
C04174=1199.785,-119.389,-38.182,179.070,5.526,149.250
C04175=1199.790,-119.639,-38.173,179.068,5.527,149.250
C04176=1199.796,-119.889,-38.163,179.066,5.526,149.251
C04177=1199.801,-120.138,-38.154,179.064,5.526,149.252
C04178=1199.806,-120.388,-38.145,179.062,5.527,149.252
C04179=1199.812,-120.638,-38.135,179.059,5.526,149.253
C04180=1199.817,-120.887,-38.126,179.058,5.526,149.253
C04181=1199.822,-121.137,-38.117,179.055,5.526,149.254
C04182=1199.828,-121.387,-38.107,179.053,5.526,149.255
C04183=1199.833,-121.637,-38.098,179.051,5.526,149.255
C04184=1199.838,-121.886,-38.089,179.049,5.526,149.256
C04185=1199.843,-122.136,-38.080,179.046,5.525,149.257
C04186=1199.849,-122.386,-38.070,179.044,5.526,149.257
C04187=1199.854,-122.636,-38.061,179.042,5.525,149.258
C04188=1199.859,-122.885,-38.052,179.040,5.525,149.258
C04189=1199.864,-123.135,-38.043,179.037,5.525,149.259
C04190=1199.870,-123.385,-38.034,179.036,5.525,149.260
C04191=1199.875,-123.635,-38.025,179.033,5.525,149.260
C04192=1199.880,-123.885,-38.015,179.031,5.525,149.261
C04193=1199.886,-124.135,-38.006,179.029,5.524,149.262
C04194=1199.891,-124.385,-37.997,179.027,5.525,149.262
C04195=1199.896,-124.634,-37.988,179.025,5.525,149.263
C04196=1199.901,-124.884,-37.979,179.022,5.524,149.264
C04197=1199.906,-125.133,-37.969,179.021,5.524,149.264
C04198=1199.912,-125.384,-37.960,179.018,5.524,149.265
C04199=1199.918,-125.633,-37.951,179.016,5.524,149.265
C04200=1199.923,-125.883,-37.942,179.014,5.523,149.266
C04201=1199.928,-126.133,-37.933,179.012,5.524,149.267
C04202=1199.934,-126.383,-37.924,179.010,5.523,149.267
C04203=1199.939,-126.632,-37.914,179.007,5.523,149.268
C04204=1199.944,-126.882,-37.905,179.005,5.523,149.269
C04205=1199.523,-126.893,-37.944,179.001,5.526,149.270
C04206=1199.518,-126.643,-37.953,179.004,5.527,149.270
C04207=1199.513,-126.393,-37.962,179.005,5.527,149.269
C04208=1199.507,-126.143,-37.971,179.008,5.527,149.269
C04209=1199.501,-125.894,-37.980,179.010,5.527,149.268
C04210=1199.496,-125.644,-37.990,179.012,5.527,149.267
C04211=1199.491,-125.395,-37.999,179.014,5.527,149.267
C04212=1199.486,-125.145,-38.007,179.016,5.528,149.266
C04213=1199.480,-124.895,-38.017,179.018,5.527,149.265
C04214=1199.475,-124.645,-38.026,179.021,5.528,149.265
C04215=1199.470,-124.396,-38.035,179.023,5.528,149.264
C04216=1199.465,-124.146,-38.044,179.025,5.528,149.263
C04217=1199.459,-123.896,-38.054,179.027,5.528,149.263
C04218=1199.454,-123.646,-38.063,179.029,5.528,149.262
C04219=1199.448,-123.396,-38.072,179.031,5.529,149.262
C04220=1199.444,-123.147,-38.081,179.033,5.528,149.261
C04221=1199.438,-122.896,-38.091,179.036,5.529,149.260
C04222=1199.432,-122.647,-38.100,179.038,5.529,149.260
C04223=1199.427,-122.397,-38.109,179.040,5.529,149.259
C04224=1199.422,-122.147,-38.118,179.042,5.529,149.259
C04225=1199.417,-121.897,-38.128,179.045,5.529,149.258
C04226=1199.411,-121.647,-38.137,179.047,5.529,149.257
C04227=1199.406,-121.398,-38.145,179.049,5.530,149.257
C04228=1199.401,-121.148,-38.156,179.051,5.529,149.256
C04229=1199.395,-120.898,-38.165,179.054,5.530,149.255
C04230=1199.390,-120.648,-38.173,179.055,5.530,149.255
C04231=1199.384,-120.398,-38.183,179.058,5.530,149.254
C04232=1199.379,-120.149,-38.193,179.060,5.530,149.254
C04233=1199.374,-119.899,-38.201,179.062,5.530,149.253
C04234=1199.369,-119.649,-38.210,179.064,5.530,149.252
C04235=1199.364,-119.400,-38.221,179.067,5.531,149.252
C04236=1199.358,-119.150,-38.229,179.069,5.530,149.251
C04237=1199.353,-118.900,-38.238,179.070,5.530,149.251
C04238=1199.348,-118.650,-38.249,179.073,5.531,149.250
C04239=1199.342,-118.401,-38.257,179.075,5.530,149.249
C04240=1199.337,-118.150,-38.267,179.077,5.531,149.249
C04241=1199.332,-117.901,-38.277,179.079,5.531,149.248
C04242=1199.327,-117.651,-38.285,179.082,5.531,149.247
C04243=1199.321,-117.402,-38.296,179.084,5.531,149.247
C04244=1199.316,-117.152,-38.305,179.086,5.532,149.246
C04245=1199.311,-116.902,-38.313,179.088,5.532,149.245
C04246=1199.305,-116.653,-38.324,179.091,5.532,149.245
C04247=1199.300,-116.403,-38.333,179.093,5.532,149.244
C04248=1199.295,-116.152,-38.342,179.095,5.532,149.244
C04249=1199.290,-115.903,-38.352,179.097,5.532,149.243
C04250=1199.284,-115.653,-38.361,179.100,5.532,149.242
C04251=1199.279,-115.403,-38.371,179.101,5.532,149.242
C04252=1199.274,-115.153,-38.380,179.104,5.533,149.241
C04253=1199.268,-114.904,-38.390,179.105,5.533,149.240
C04254=1199.263,-114.654,-38.399,179.108,5.533,149.240
C04255=1199.258,-114.404,-38.408,179.110,5.533,149.239
C04256=1199.252,-114.155,-38.418,179.112,5.534,149.239
C04257=1199.247,-113.905,-38.427,179.114,5.533,149.238
C04258=1199.241,-113.655,-38.437,179.117,5.534,149.237
C04259=1199.236,-113.405,-38.446,179.119,5.534,149.237
C04260=1199.231,-113.156,-38.456,179.121,5.534,149.236
C04261=1199.226,-112.905,-38.466,179.124,5.534,149.235
C04262=1199.221,-112.656,-38.476,179.126,5.534,149.235
C04263=1199.215,-112.406,-38.485,179.128,5.534,149.234
C04264=1199.210,-112.156,-38.495,179.130,5.534,149.233
C04265=1199.205,-111.906,-38.504,179.132,5.534,149.233
C04266=1199.200,-111.657,-38.514,179.135,5.535,149.232
C04267=1199.194,-111.407,-38.523,179.136,5.535,149.232
C04268=1199.189,-111.158,-38.533,179.139,5.535,149.231
C04269=1199.183,-110.908,-38.542,179.141,5.535,149.230
C04270=1199.179,-110.658,-38.552,179.143,5.536,149.230
C04271=1199.173,-110.408,-38.562,179.145,5.535,149.229
C04272=1199.168,-110.158,-38.571,179.148,5.536,149.228
C04273=1199.162,-109.909,-38.581,179.150,5.536,149.228
C04274=1199.157,-109.659,-38.590,179.152,5.536,149.227
C04275=1199.152,-109.409,-38.601,179.154,5.536,149.226
C04276=1199.146,-109.159,-38.610,179.157,5.536,149.226
C04277=1199.141,-108.909,-38.620,179.159,5.536,149.225
C04278=1199.136,-108.660,-38.630,179.161,5.536,149.224
C04279=1199.131,-108.410,-38.639,179.163,5.536,149.224
C04280=1199.125,-108.160,-38.649,179.166,5.537,149.223
C04281=1199.120,-107.911,-38.658,179.168,5.536,149.222
C04282=1199.114,-107.661,-38.668,179.170,5.537,149.222
C04283=1199.110,-107.411,-38.678,179.172,5.537,149.221
C04284=1199.104,-107.161,-38.688,179.175,5.537,149.221
C04285=1199.099,-106.912,-38.698,179.176,5.537,149.220
C04286=1199.094,-106.662,-38.708,179.179,5.538,149.219
C04287=1199.088,-106.412,-38.717,179.181,5.537,149.219
C04288=1199.084,-106.162,-38.727,179.183,5.538,149.218
C04289=1199.078,-105.912,-38.737,179.185,5.538,149.217
C04290=1199.073,-105.663,-38.746,179.188,5.538,149.217
C04291=1199.067,-105.413,-38.757,179.190,5.538,149.216
C04292=1199.062,-105.164,-38.767,179.192,5.538,149.216
C04293=1199.057,-104.913,-38.776,179.194,5.538,149.215
C04294=1199.051,-104.663,-38.786,179.197,5.539,149.214
C04295=1199.047,-104.414,-38.796,179.199,5.538,149.214
C04296=1199.041,-104.165,-38.806,179.201,5.539,149.213
C04297=1199.035,-103.915,-38.816,179.203,5.539,149.212
C04298=1199.031,-103.665,-38.825,179.206,5.539,149.212
C04299=1199.025,-103.415,-38.836,179.208,5.539,149.211
C04300=1199.020,-103.166,-38.845,179.210,5.539,149.210
C04301=1199.014,-102.916,-38.855,179.212,5.539,149.210
C04302=1199.009,-102.665,-38.865,179.215,5.540,149.209
C04303=1199.005,-102.416,-38.875,179.217,5.539,149.208
C04304=1198.999,-102.167,-38.885,179.219,5.540,149.208
C04305=1198.993,-101.916,-38.895,179.221,5.540,149.207
C04306=1198.988,-101.645,-38.906,179.224,5.540,149.206
C04307=1198.983,-101.374,-38.917,179.226,5.540,149.206
C04308=1198.976,-101.102,-38.927,179.228,5.540,149.205
C04309=1198.971,-100.831,-38.938,179.231,5.540,149.204
C04310=1198.966,-100.581,-38.949,179.233,5.541,149.204
C04311=1198.960,-100.331,-38.959,179.235,5.541,149.203
C04312=1198.955,-100.082,-38.968,179.238,5.541,149.202
C04313=1198.949,-99.832,-38.978,179.240,5.541,149.202
C04314=1198.944,-99.582,-38.988,179.242,5.542,149.201
C04315=1198.939,-99.332,-38.998,179.244,5.541,149.201
C04316=1198.934,-99.083,-39.008,179.247,5.542,149.200
C04317=1198.928,-98.833,-39.018,179.249,5.542,149.199
C04318=1198.923,-98.583,-39.029,179.251,5.542,149.199
C04319=1198.918,-98.334,-39.039,179.253,5.542,149.198
C04320=1198.913,-98.084,-39.049,179.256,5.542,149.197
C04321=1198.908,-97.833,-39.059,179.258,5.542,149.197
C04322=1198.902,-97.584,-39.069,179.260,5.543,149.196
C04323=1198.897,-97.335,-39.079,179.262,5.543,149.196
C04324=1198.892,-97.084,-39.089,179.265,5.543,149.195
C04325=1198.886,-96.835,-39.099,179.267,5.543,149.194
C04326=1198.881,-96.585,-39.110,179.269,5.543,149.193
C04327=1198.876,-96.336,-39.119,179.272,5.544,149.193
C04328=1198.871,-96.086,-39.130,179.274,5.543,149.192
C04329=1198.865,-95.836,-39.140,179.276,5.544,149.191
C04330=1198.860,-95.587,-39.150,179.278,5.544,149.191
C04331=1198.855,-95.337,-39.161,179.281,5.544,149.190
C04332=1198.850,-95.087,-39.170,179.283,5.544,149.190
C04333=1198.844,-94.838,-39.181,179.285,5.545,149.189
C04334=1198.839,-94.587,-39.191,179.287,5.544,149.188
C04335=1198.834,-94.338,-39.201,179.290,5.545,149.188
C04336=1198.828,-94.088,-39.212,179.292,5.544,149.187
C04337=1198.824,-93.838,-39.222,179.294,5.545,149.186
C04338=1198.818,-93.589,-39.232,179.297,5.545,149.186
C04339=1198.813,-93.339,-39.242,179.299,5.545,149.185
C04340=1198.808,-93.089,-39.253,179.301,5.546,149.185
C04341=1198.802,-92.840,-39.263,179.303,5.546,149.184
C04342=1198.797,-92.589,-39.273,179.306,5.546,149.183
C04343=1198.792,-92.340,-39.283,179.308,5.546,149.182
C04344=1198.787,-92.091,-39.293,179.310,5.546,149.182
C04345=1198.782,-91.840,-39.304,179.312,5.546,149.181
C04346=1198.776,-91.591,-39.314,179.315,5.546,149.181
C04347=1198.771,-91.341,-39.324,179.317,5.546,149.180
C04348=1198.765,-91.091,-39.335,179.319,5.547,149.179
C04349=1198.760,-90.841,-39.345,179.322,5.547,149.179
C04350=1198.755,-90.591,-39.355,179.324,5.547,149.178
C04351=1198.750,-90.342,-39.365,179.326,5.548,149.177
C04352=1198.744,-90.092,-39.375,179.328,5.547,149.177
C04353=1198.739,-89.842,-39.386,179.331,5.548,149.176
C04354=1198.734,-89.593,-39.397,179.333,5.547,149.175
C04355=1198.729,-89.343,-39.407,179.335,5.548,149.175
C04356=1198.724,-89.093,-39.418,179.337,5.548,149.174
C04357=1198.719,-88.843,-39.428,179.340,5.548,149.173
C04358=1198.713,-88.594,-39.438,179.342,5.549,149.173
C04359=1198.707,-88.344,-39.449,179.344,5.549,149.172
C04360=1198.702,-88.094,-39.459,179.347,5.549,149.171
C04361=1198.697,-87.845,-39.470,179.349,5.549,149.171
C04362=1198.692,-87.595,-39.481,179.351,5.549,149.170
C04363=1198.687,-87.346,-39.490,179.353,5.549,149.170
C04364=1198.682,-87.095,-39.501,179.356,5.549,149.169
C04365=1198.677,-86.846,-39.511,179.358,5.549,149.168
C04366=1198.672,-86.596,-39.522,179.360,5.550,149.168
C04367=1198.666,-86.347,-39.533,179.363,5.550,149.167
C04368=1198.661,-86.097,-39.543,179.365,5.550,149.166
C04369=1198.656,-85.847,-39.553,179.367,5.550,149.166
C04370=1198.650,-85.597,-39.564,179.369,5.550,149.165
C04371=1198.645,-85.348,-39.575,179.372,5.551,149.164
C04372=1198.640,-85.098,-39.585,179.374,5.550,149.164
C04373=1198.635,-84.848,-39.596,179.376,5.551,149.163
C04374=1198.629,-84.598,-39.606,179.379,5.552,149.162
C04375=1198.625,-84.349,-39.617,179.381,5.551,149.162
C04376=1198.619,-84.099,-39.627,179.383,5.552,149.161
C04377=1198.614,-83.849,-39.638,179.385,5.551,149.160
C04378=1198.608,-83.599,-39.648,179.388,5.552,149.160
C04379=1198.604,-83.350,-39.659,179.390,5.552,149.159
C04380=1198.598,-83.100,-39.670,179.392,5.552,149.158
C04381=1198.593,-82.850,-39.680,179.395,5.553,149.158
C04382=1198.588,-82.601,-39.691,179.397,5.553,149.157
C04383=1198.583,-82.351,-39.702,179.399,5.553,149.157
C04384=1198.577,-82.101,-39.712,179.401,5.553,149.156
C04385=1198.572,-81.851,-39.724,179.404,5.553,149.155
C04386=1198.566,-81.602,-39.734,179.406,5.553,149.155
C04387=1198.561,-81.351,-39.745,179.408,5.553,149.154
C04388=1198.556,-81.103,-39.755,179.411,5.554,149.153
C04389=1198.551,-80.852,-39.766,179.413,5.554,149.153
C04390=1198.545,-80.603,-39.776,179.415,5.554,149.152
C04391=1198.541,-80.353,-39.788,179.417,5.554,149.151
C04392=1198.535,-80.104,-39.798,179.420,5.554,149.151
C04393=1198.530,-79.854,-39.809,179.422,5.555,149.150
C04394=1198.525,-79.604,-39.819,179.424,5.555,149.149
C04395=1198.520,-79.354,-39.830,179.427,5.555,149.149
C04396=1198.514,-79.104,-39.842,179.429,5.555,149.148
C04397=1198.509,-78.855,-39.852,179.432,5.555,149.147
C04398=1198.504,-78.605,-39.863,179.433,5.555,149.147
C04399=1198.498,-78.356,-39.873,179.436,5.556,149.146
C04400=1198.493,-78.105,-39.884,179.439,5.556,149.145
C04401=1198.488,-77.856,-39.895,179.441,5.556,149.145
C04402=1198.483,-77.606,-39.905,179.443,5.557,149.144
C04403=1198.478,-77.356,-39.917,179.445,5.556,149.143
C04404=1198.472,-77.107,-39.928,179.448,5.557,149.143
C04405=1198.467,-76.857,-39.939,179.450,5.557,149.142
C04406=1198.462,-76.607,-39.949,179.452,5.557,149.142
C04407=1198.457,-76.358,-39.960,179.455,5.557,149.141
C04408=1198.451,-76.108,-39.971,179.457,5.557,149.140
C04409=1198.446,-75.858,-39.982,179.459,5.558,149.139
C04410=1198.441,-75.587,-39.993,179.462,5.558,149.139
C04411=1198.435,-75.317,-40.005,179.464,5.558,149.138
C04412=1198.429,-75.046,-40.018,179.467,5.558,149.137
C04413=1198.424,-74.775,-40.029,179.470,5.558,149.137
C04414=1198.418,-74.525,-40.040,179.472,5.559,149.136
C04415=1198.413,-74.276,-40.051,179.474,5.559,149.135
C04416=1198.408,-74.027,-40.062,179.476,5.559,149.135
C04417=1198.403,-73.776,-40.073,179.479,5.559,149.134
C04418=1198.397,-73.527,-40.085,179.481,5.560,149.134
C04419=1198.392,-73.277,-40.095,179.483,5.560,149.133
C04420=1198.387,-73.027,-40.106,179.486,5.560,149.132
C04421=1198.381,-72.778,-40.116,179.488,5.560,149.131
C04422=1198.376,-72.528,-40.128,179.490,5.560,149.131
C04423=1198.371,-72.278,-40.140,179.492,5.561,149.130
C04424=1198.366,-72.029,-40.150,179.495,5.561,149.130
C04425=1198.361,-71.779,-40.161,179.497,5.561,149.129
C04426=1198.355,-71.529,-40.172,179.500,5.561,149.128
C04427=1198.350,-71.280,-40.183,179.501,5.561,149.128
C04428=1198.345,-71.030,-40.194,179.504,5.562,149.127
C04429=1198.340,-70.780,-40.205,179.507,5.562,149.126
C04430=1198.334,-70.531,-40.217,179.509,5.562,149.125
C04431=1198.330,-70.281,-40.228,179.512,5.562,149.125
C04432=1198.325,-70.031,-40.238,179.513,5.562,149.124
C04433=1198.319,-69.781,-40.250,179.516,5.563,149.124
C04434=1198.314,-69.532,-40.261,179.519,5.563,149.123
C04435=1198.309,-69.282,-40.272,179.521,5.563,149.122
C04436=1198.303,-69.032,-40.283,179.523,5.563,149.122
C04437=1198.298,-68.783,-40.295,179.525,5.564,149.121
C04438=1198.293,-68.532,-40.305,179.528,5.563,149.120
C04439=1198.287,-68.283,-40.317,179.530,5.564,149.120
C04440=1198.282,-68.034,-40.328,179.532,5.564,149.119
C04441=1198.277,-67.783,-40.339,179.534,5.564,149.118
C04442=1198.272,-67.533,-40.350,179.537,5.565,149.118
C04443=1198.267,-67.284,-40.361,179.539,5.564,149.117
C04444=1198.262,-67.035,-40.373,179.542,5.565,149.116
C04445=1198.256,-66.784,-40.384,179.544,5.566,149.116
C04446=1198.251,-66.535,-40.395,179.546,5.565,149.115
C04447=1198.246,-66.286,-40.406,179.549,5.566,149.114
C04448=1198.241,-66.036,-40.418,179.551,5.565,149.114
C04449=1198.236,-65.786,-40.429,179.554,5.566,149.113
C04450=1198.230,-65.536,-40.440,179.556,5.567,149.113
C04451=1198.225,-65.287,-40.451,179.558,5.566,149.112
C04452=1198.221,-65.037,-40.463,179.560,5.567,149.111
C04453=1198.215,-64.787,-40.474,179.563,5.567,149.110
C04454=1198.210,-64.538,-40.485,179.565,5.567,149.110
C04455=1198.204,-64.288,-40.497,179.567,5.568,149.109
C04456=1198.199,-64.038,-40.508,179.570,5.567,149.109
C04457=1198.194,-63.788,-40.520,179.572,5.568,149.108
C04458=1198.189,-63.539,-40.531,179.575,5.568,149.107
C04459=1198.184,-63.290,-40.542,179.576,5.568,149.107
C04460=1198.179,-63.040,-40.554,179.579,5.569,149.106
C04461=1198.174,-62.789,-40.564,179.582,5.569,149.105
C04462=1198.167,-62.540,-40.576,179.584,5.569,149.104
C04463=1198.163,-62.290,-40.587,179.587,5.569,149.104
C04464=1198.157,-62.041,-40.599,179.589,5.570,149.103
C04465=1198.153,-61.791,-40.610,179.591,5.570,149.103
C04466=1198.147,-61.541,-40.622,179.593,5.570,149.102
C04467=1198.142,-61.292,-40.633,179.596,5.570,149.101
C04468=1198.137,-61.042,-40.645,179.598,5.570,149.100
C04469=1198.132,-60.793,-40.656,179.600,5.571,149.100
C04470=1198.127,-60.543,-40.668,179.602,5.570,149.099
C04471=1198.122,-60.293,-40.680,179.605,5.571,149.099
C04472=1198.116,-60.044,-40.690,179.608,5.571,149.098
C04473=1198.111,-59.793,-40.702,179.610,5.571,149.097
C04474=1198.106,-59.544,-40.713,179.612,5.572,149.097
C04475=1198.101,-59.294,-40.725,179.615,5.572,149.096
C04476=1198.095,-59.044,-40.737,179.617,5.572,149.095
C04477=1198.090,-58.795,-40.748,179.619,5.572,149.095
C04478=1198.084,-58.545,-40.760,179.622,5.573,149.094
C04479=1198.080,-58.295,-40.771,179.624,5.573,149.093
C04480=1198.074,-58.046,-40.783,179.626,5.573,149.093
C04481=1198.070,-57.796,-40.794,179.629,5.574,149.092
C04482=1198.064,-57.546,-40.806,179.631,5.573,149.091
C04483=1198.059,-57.296,-40.817,179.634,5.574,149.091
C04484=1198.053,-57.047,-40.829,179.636,5.575,149.090
C04485=1198.049,-56.798,-40.841,179.638,5.574,149.089
C04486=1198.044,-56.548,-40.853,179.641,5.575,149.089
C04487=1198.038,-56.298,-40.864,179.643,5.575,149.088
C04488=1198.034,-56.049,-40.876,179.646,5.575,149.087
C04489=1198.028,-55.799,-40.888,179.648,5.576,149.087
C04490=1198.023,-55.549,-40.899,179.650,5.576,149.086
C04491=1198.017,-55.300,-40.910,179.652,5.576,149.085
C04492=1198.013,-55.050,-40.922,179.655,5.576,149.085
C04493=1198.007,-54.800,-40.934,179.658,5.577,149.084
C04494=1198.002,-54.550,-40.945,179.659,5.577,149.084
C04495=1197.997,-54.301,-40.957,179.662,5.577,149.083
C04496=1197.992,-54.051,-40.969,179.665,5.577,149.082
C04497=1197.987,-53.801,-40.981,179.667,5.577,149.081
C04498=1197.982,-53.552,-40.993,179.669,5.578,149.081
C04499=1197.976,-53.302,-41.004,179.672,5.578,149.080
C04500=1197.972,-53.052,-41.016,179.674,5.578,149.080
C04501=1197.966,-52.802,-41.028,179.676,5.578,149.079
C04502=1197.960,-52.553,-41.039,179.679,5.579,149.078
C04503=1197.956,-52.304,-41.051,179.681,5.579,149.077
C04504=1197.950,-52.054,-41.063,179.683,5.579,149.077
C04505=1197.945,-51.804,-41.075,179.686,5.580,149.076
C04506=1197.940,-51.555,-41.086,179.688,5.579,149.076
C04507=1197.935,-51.305,-41.098,179.691,5.580,149.075
C04508=1197.930,-51.055,-41.111,179.693,5.580,149.074
C04509=1197.925,-50.806,-41.122,179.695,5.580,149.074
C04510=1197.920,-50.556,-41.134,179.698,5.581,149.073
C04511=1197.914,-50.306,-41.146,179.700,5.581,149.072
C04512=1197.909,-50.056,-41.158,179.702,5.581,149.072
C04513=1197.904,-49.807,-41.170,179.705,5.581,149.071
C04514=1197.899,-49.537,-41.182,179.708,5.582,149.070
C04515=1197.893,-49.267,-41.195,179.710,5.582,149.069
C04516=1197.887,-48.996,-41.209,179.713,5.583,149.069
C04517=1197.881,-48.727,-41.221,179.715,5.582,149.068
C04518=1197.877,-48.477,-41.233,179.718,5.583,149.067
C04519=1197.871,-48.227,-41.245,179.720,5.584,149.067
C04520=1197.866,-47.977,-41.256,179.722,5.583,149.066
C04521=1197.861,-47.728,-41.269,179.725,5.584,149.065
C04522=1197.856,-47.478,-41.280,179.727,5.584,149.065
C04523=1197.850,-47.228,-41.292,179.730,5.585,149.064
C04524=1197.845,-46.979,-41.305,179.732,5.585,149.064
C04525=1197.840,-46.729,-41.317,179.734,5.585,149.063
C04526=1197.834,-46.479,-41.329,179.737,5.586,149.062
C04527=1197.830,-46.230,-41.341,179.739,5.585,149.061
C04528=1197.825,-45.980,-41.352,179.742,5.586,149.061
C04529=1197.819,-45.730,-41.364,179.744,5.586,149.060
C04530=1197.814,-45.481,-41.377,179.746,5.586,149.060
C04531=1197.809,-45.231,-41.389,179.749,5.587,149.059
C04532=1197.804,-44.982,-41.401,179.751,5.587,149.058
C04533=1197.799,-44.732,-41.413,179.754,5.588,149.057
C04534=1197.793,-44.482,-41.425,179.756,5.587,149.057
C04535=1197.788,-44.233,-41.437,179.758,5.588,149.056
C04536=1197.783,-43.983,-41.449,179.761,5.588,149.056
C04537=1197.778,-43.733,-41.462,179.763,5.588,149.055
C04538=1197.773,-43.484,-41.473,179.766,5.589,149.054
C04539=1197.768,-43.234,-41.486,179.768,5.589,149.054
C04540=1197.763,-42.985,-41.497,179.770,5.589,149.053
C04541=1197.758,-42.734,-41.510,179.773,5.589,149.052
C04542=1197.753,-42.485,-41.522,179.775,5.590,149.052
C04543=1197.747,-42.235,-41.534,179.778,5.590,149.051
C04544=1197.742,-41.985,-41.547,179.780,5.590,149.050
C04545=1197.737,-41.735,-41.559,179.783,5.590,149.050
C04546=1197.732,-41.486,-41.571,179.785,5.591,149.049
C04547=1197.727,-41.236,-41.583,179.787,5.592,149.048
C04548=1197.722,-40.987,-41.595,179.790,5.591,149.048
C04549=1197.716,-40.737,-41.607,179.792,5.592,149.047
C04550=1197.711,-40.488,-41.620,179.795,5.592,149.046
C04551=1197.706,-40.238,-41.632,179.796,5.592,149.046
C04552=1197.701,-39.989,-41.644,179.799,5.593,149.045
C04553=1197.695,-39.739,-41.657,179.802,5.593,149.044
C04554=1197.691,-39.489,-41.669,179.804,5.594,149.044
C04555=1197.685,-39.239,-41.682,179.807,5.593,149.043
C04556=1197.680,-38.989,-41.694,179.809,5.594,149.043
C04557=1197.675,-38.740,-41.706,179.811,5.595,149.042
C04558=1197.669,-38.490,-41.718,179.813,5.594,149.041
C04559=1197.664,-38.241,-41.731,179.816,5.595,149.040
C04560=1197.659,-37.992,-41.743,179.819,5.595,149.040
C04561=1197.654,-37.742,-41.755,179.821,5.596,149.039
C04562=1197.649,-37.492,-41.768,179.823,5.596,149.039
C04563=1197.644,-37.242,-41.780,179.826,5.596,149.038
C04564=1197.639,-36.992,-41.793,179.828,5.597,149.037
C04565=1197.634,-36.743,-41.805,179.831,5.597,149.036
C04566=1197.628,-36.493,-41.817,179.833,5.597,149.036
C04567=1197.623,-36.244,-41.830,179.835,5.598,149.035
C04568=1197.618,-35.994,-41.842,179.838,5.598,149.035
C04569=1197.612,-35.744,-41.854,179.841,5.599,149.034
C04570=1197.608,-35.494,-41.867,179.843,5.598,149.033
C04571=1197.603,-35.245,-41.880,179.845,5.599,149.032
C04572=1197.597,-34.995,-41.892,179.848,5.599,149.032
C04573=1197.592,-34.746,-41.904,179.850,5.599,149.031
C04574=1197.587,-34.497,-41.917,179.852,5.600,149.031
C04575=1197.582,-34.247,-41.929,179.855,5.600,149.030
C04576=1197.577,-33.997,-41.942,179.858,5.601,149.029
C04577=1197.572,-33.747,-41.954,179.860,5.600,149.029
C04578=1197.567,-33.498,-41.967,179.862,5.601,149.028
C04579=1197.562,-33.248,-41.979,179.865,5.601,149.027
C04580=1197.556,-32.999,-41.991,179.867,5.602,149.027
C04581=1197.551,-32.749,-42.004,179.869,5.602,149.026
C04582=1197.547,-32.499,-42.017,179.872,5.602,149.025
C04583=1197.541,-32.249,-42.029,179.875,5.602,149.025
C04584=1197.536,-32.000,-42.041,179.877,5.603,149.024
C04585=1197.530,-31.750,-42.055,179.879,5.603,149.023
C04586=1197.526,-31.500,-42.068,179.881,5.603,149.023
C04587=1197.520,-31.251,-42.079,179.884,5.604,149.022
C04588=1197.515,-31.001,-42.092,179.887,5.604,149.021
C04589=1197.510,-30.752,-42.105,179.889,5.605,149.021
C04590=1197.505,-30.503,-42.117,179.891,5.605,149.020
C04591=1197.501,-30.253,-42.130,179.894,5.605,149.019
C04592=1197.495,-30.003,-42.143,179.896,5.606,149.019
C04593=1197.489,-29.753,-42.155,179.899,5.606,149.018
C04594=1197.484,-29.504,-42.168,179.901,5.606,149.017
C04595=1197.480,-29.254,-42.181,179.903,5.607,149.017
C04596=1197.474,-29.004,-42.193,179.906,5.607,149.016
C04597=1197.469,-28.755,-42.206,179.909,5.608,149.015
C04598=1197.464,-28.506,-42.219,179.911,5.607,149.015
C04599=1197.459,-28.255,-42.232,179.913,5.608,149.014
C04600=1197.454,-28.006,-42.245,179.916,5.608,149.013
C04601=1197.448,-27.756,-42.257,179.918,5.609,149.013
C04602=1197.443,-27.507,-42.269,179.920,5.609,149.012
C04603=1197.439,-27.257,-42.282,179.923,5.609,149.012
C04604=1197.433,-27.007,-42.295,179.926,5.610,149.011
C04605=1197.428,-26.758,-42.308,179.928,5.610,149.010
C04606=1197.423,-26.508,-42.321,179.930,5.611,149.010
C04607=1197.418,-26.259,-42.334,179.933,5.611,149.009
C04608=1197.413,-26.009,-42.346,179.935,5.611,149.008
C04609=1197.407,-25.760,-42.359,179.938,5.612,149.008
C04610=1197.403,-25.510,-42.372,179.940,5.612,149.007
C04611=1197.397,-25.260,-42.385,179.943,5.612,149.006
C04612=1197.392,-25.011,-42.398,179.945,5.613,149.006
C04613=1197.387,-24.761,-42.411,179.947,5.613,149.005
C04614=1197.382,-24.511,-42.424,179.950,5.614,149.004
C04615=1197.377,-24.262,-42.436,179.953,5.614,149.004
C04616=1197.372,-24.012,-42.449,179.955,5.614,149.003
C04617=1197.366,-23.762,-42.462,179.957,5.615,149.002
C04618=1197.361,-23.493,-42.476,179.960,5.615,149.002
C04619=1197.355,-23.223,-42.490,179.963,5.615,149.001
C04620=1197.350,-22.954,-42.504,179.965,5.616,149.000
C04621=1197.345,-22.684,-42.519,179.968,5.616,148.999
C04622=1197.340,-22.435,-42.531,179.970,5.617,148.999
C04623=1197.334,-22.185,-42.544,179.973,5.617,148.998
C04624=1197.329,-21.935,-42.558,179.975,5.617,148.998
C04625=1197.324,-21.686,-42.570,179.978,5.617,148.997
C04626=1197.319,-21.436,-42.583,179.980,5.618,148.996
C04627=1197.314,-21.186,-42.596,179.983,5.618,148.995
C04628=1197.309,-20.937,-42.609,179.985,5.619,148.995
C04629=1197.304,-20.687,-42.622,179.987,5.619,148.994
C04630=1197.298,-20.437,-42.635,179.990,5.619,148.994
C04631=1197.293,-20.189,-42.648,179.993,5.620,148.993
C04632=1197.289,-19.938,-42.661,179.995,5.620,148.992
C04633=1197.283,-19.689,-42.675,179.997,5.621,148.992
C04634=1197.278,-19.440,-42.687,179.999,5.621,148.991
C04635=1197.273,-19.189,-42.701,-179.998,5.621,148.990
C04636=1197.267,-18.940,-42.713,-179.995,5.622,148.990
C04637=1197.263,-18.690,-42.727,-179.993,5.622,148.989
C04638=1197.257,-18.441,-42.740,-179.990,5.623,148.988
C04639=1197.252,-18.192,-42.753,-179.988,5.623,148.988
C04640=1197.247,-17.941,-42.766,-179.986,5.623,148.987
C04641=1197.242,-17.692,-42.779,-179.983,5.624,148.986
C04642=1197.238,-17.442,-42.793,-179.980,5.624,148.986
C04643=1197.232,-17.193,-42.806,-179.978,5.625,148.985
C04644=1197.227,-16.943,-42.819,-179.976,5.625,148.985
C04645=1197.221,-16.693,-42.832,-179.973,5.625,148.984
C04646=1197.217,-16.445,-42.845,-179.971,5.626,148.983
C04647=1197.211,-16.194,-42.859,-179.968,5.626,148.983
C04648=1197.206,-15.945,-42.871,-179.965,5.627,148.982
C04649=1197.202,-15.695,-42.884,-179.963,5.627,148.981
C04650=1197.196,-15.446,-42.898,-179.961,5.627,148.981
C04651=1197.192,-15.196,-42.911,-179.959,5.628,148.980
C04652=1197.186,-14.946,-42.924,-179.956,5.628,148.979
C04653=1197.182,-14.697,-42.938,-179.953,5.629,148.979
C04654=1197.176,-14.447,-42.951,-179.951,5.629,148.978
C04655=1197.171,-14.198,-42.964,-179.948,5.630,148.977
C04656=1197.166,-13.948,-42.978,-179.946,5.630,148.977
C04657=1197.160,-13.699,-42.991,-179.944,5.630,148.976
C04658=1197.155,-13.448,-43.004,-179.941,5.631,148.975
C04659=1197.150,-13.200,-43.018,-179.938,5.631,148.975
C04660=1197.145,-12.949,-43.031,-179.936,5.631,148.974
C04661=1197.140,-12.700,-43.044,-179.934,5.632,148.973
C04662=1197.135,-12.450,-43.058,-179.931,5.632,148.973
C04663=1197.130,-12.201,-43.071,-179.929,5.632,148.972
C04664=1197.125,-11.951,-43.085,-179.926,5.633,148.971
C04665=1197.120,-11.702,-43.098,-179.923,5.633,148.971
C04666=1197.115,-11.452,-43.111,-179.921,5.634,148.970
C04667=1197.109,-11.203,-43.125,-179.919,5.635,148.970
C04668=1197.104,-10.953,-43.138,-179.917,5.634,148.969
C04669=1197.099,-10.704,-43.152,-179.914,5.635,148.968
C04670=1197.094,-10.454,-43.165,-179.911,5.635,148.967
C04671=1197.089,-10.205,-43.179,-179.909,5.636,148.967
C04672=1197.084,-9.955,-43.192,-179.906,5.637,148.966
C04673=1197.079,-9.705,-43.206,-179.904,5.637,148.966
C04674=1197.074,-9.455,-43.219,-179.902,5.637,148.965
C04675=1197.069,-9.205,-43.232,-179.899,5.637,148.964
C04676=1197.063,-8.956,-43.246,-179.896,5.638,148.964
C04677=1197.059,-8.706,-43.259,-179.894,5.639,148.963
C04678=1197.053,-8.457,-43.273,-179.892,5.639,148.962
C04679=1197.048,-8.208,-43.287,-179.889,5.640,148.962
C04680=1197.043,-7.958,-43.300,-179.886,5.640,148.961
C04681=1197.038,-7.709,-43.314,-179.884,5.640,148.960
C04682=1197.034,-7.459,-43.327,-179.882,5.641,148.960
C04683=1197.028,-7.210,-43.341,-179.879,5.641,148.959
C04684=1197.023,-6.959,-43.355,-179.877,5.642,148.959
C04685=1197.018,-6.710,-43.368,-179.874,5.642,148.958
C04686=1197.013,-6.460,-43.382,-179.871,5.643,148.957
C04687=1197.007,-6.211,-43.395,-179.869,5.643,148.956
C04688=1197.003,-5.962,-43.409,-179.867,5.643,148.956
C04689=1196.998,-5.711,-43.423,-179.865,5.644,148.955
C04690=1196.992,-5.462,-43.437,-179.862,5.644,148.955
C04691=1196.988,-5.212,-43.450,-179.859,5.645,148.954
C04692=1196.982,-4.963,-43.463,-179.857,5.645,148.953
C04693=1196.977,-4.714,-43.478,-179.854,5.646,148.953
C04694=1196.972,-4.463,-43.491,-179.852,5.646,148.952
C04695=1196.967,-4.215,-43.505,-179.849,5.647,148.951
C04696=1196.962,-3.965,-43.519,-179.847,5.647,148.951
C04697=1196.956,-3.715,-43.532,-179.844,5.647,148.950
C04698=1196.952,-3.466,-43.546,-179.842,5.648,148.950
C04699=1196.947,-3.216,-43.560,-179.840,5.648,148.949
C04700=1196.941,-2.967,-43.573,-179.837,5.649,148.948
C04701=1196.936,-2.717,-43.588,-179.834,5.649,148.947
C04702=1196.932,-2.467,-43.601,-179.832,5.650,148.947
C04703=1196.926,-2.218,-43.614,-179.829,5.651,148.946
C04704=1196.921,-1.968,-43.629,-179.827,5.650,148.946
C04705=1196.916,-1.718,-43.643,-179.825,5.651,148.945
C04706=1196.911,-1.469,-43.656,-179.822,5.651,148.944
C04707=1196.906,-1.219,-43.670,-179.819,5.652,148.944
C04708=1196.901,-0.970,-43.684,-179.817,5.653,148.943
C04709=1196.896,-0.721,-43.698,-179.815,5.653,148.942
C04710=1196.891,-0.470,-43.712,-179.812,5.654,148.942
C04711=1196.886,-0.221,-43.725,-179.809,5.654,148.941
C04712=1196.881,0.028,-43.739,-179.807,5.655,148.940
C04713=1196.876,0.278,-43.753,-179.805,5.655,148.940
C04714=1196.871,0.528,-43.768,-179.802,5.655,148.939
C04715=1196.865,0.777,-43.781,-179.800,5.656,148.938
C04716=1196.860,1.027,-43.795,-179.797,5.656,148.938
C04717=1196.856,1.276,-43.809,-179.794,5.657,148.937
C04718=1196.850,1.525,-43.823,-179.792,5.657,148.936
C04719=1196.845,1.775,-43.837,-179.790,5.658,148.936
C04720=1196.840,2.025,-43.851,-179.787,5.659,148.935
C04721=1196.835,2.275,-43.865,-179.784,5.659,148.935
C04722=1196.829,2.543,-43.880,-179.782,5.659,148.934
C04723=1196.824,2.813,-43.895,-179.779,5.660,148.933
C04724=1196.819,3.082,-43.910,-179.776,5.660,148.933
C04725=1196.813,3.351,-43.925,-179.774,5.661,148.932
C04726=1196.808,3.600,-43.939,-179.771,5.661,148.931
C04727=1196.803,3.850,-43.953,-179.768,5.662,148.930
C04728=1196.798,4.100,-43.968,-179.766,5.663,148.930
C04729=1196.793,4.349,-43.981,-179.764,5.663,148.929
C04730=1196.788,4.598,-43.995,-179.761,5.663,148.929
C04731=1196.783,4.848,-44.010,-179.759,5.663,148.928
C04732=1196.778,5.098,-44.024,-179.756,5.664,148.927
C04733=1196.773,5.347,-44.038,-179.754,5.665,148.927
C04734=1196.767,5.596,-44.052,-179.751,5.665,148.926
C04735=1196.762,5.846,-44.066,-179.749,5.666,148.925
C04736=1196.758,6.096,-44.081,-179.746,5.666,148.925
C04737=1196.753,6.345,-44.095,-179.743,5.667,148.924
C04738=1196.748,6.595,-44.109,-179.741,5.668,148.924
C04739=1196.742,6.844,-44.123,-179.739,5.668,148.923
C04740=1196.737,7.094,-44.137,-179.736,5.669,148.922
C04741=1196.732,7.344,-44.152,-179.733,5.669,148.922
C04742=1196.727,7.593,-44.166,-179.731,5.670,148.921
C04743=1196.722,7.843,-44.180,-179.729,5.670,148.920
C04744=1196.717,8.092,-44.194,-179.726,5.670,148.920
C04745=1196.712,8.342,-44.208,-179.724,5.671,148.919
C04746=1196.707,8.591,-44.223,-179.721,5.671,148.918
C04747=1196.702,8.841,-44.237,-179.719,5.672,148.918
C04748=1196.697,9.091,-44.251,-179.716,5.673,148.917
C04749=1196.691,9.340,-44.265,-179.714,5.673,148.917
C04750=1196.686,9.590,-44.279,-179.711,5.674,148.916
C04751=1196.681,9.839,-44.294,-179.708,5.674,148.915
C04752=1196.676,10.089,-44.308,-179.706,5.675,148.915
C04753=1196.672,10.338,-44.323,-179.703,5.675,148.914
C04754=1196.667,10.588,-44.337,-179.701,5.676,148.913
C04755=1196.661,10.837,-44.351,-179.698,5.676,148.913
C04756=1196.656,11.087,-44.365,-179.696,5.677,148.912
C04757=1196.651,11.336,-44.380,-179.693,5.678,148.911
C04758=1196.646,11.586,-44.394,-179.691,5.678,148.911
C04759=1196.641,11.836,-44.408,-179.689,5.678,148.910
C04760=1196.637,12.085,-44.423,-179.686,5.678,148.909
C04761=1196.632,12.334,-44.437,-179.683,5.679,148.909
C04762=1196.626,12.584,-44.452,-179.681,5.680,148.908
C04763=1196.621,12.833,-44.466,-179.679,5.680,148.908
C04764=1196.616,13.083,-44.481,-179.676,5.681,148.907
C04765=1196.611,13.332,-44.496,-179.673,5.681,148.906
C04766=1196.606,13.582,-44.510,-179.671,5.682,148.906
C04767=1196.601,13.832,-44.524,-179.668,5.683,148.905
C04768=1196.596,14.081,-44.538,-179.666,5.683,148.904
C04769=1196.592,14.331,-44.553,-179.663,5.684,148.904
C04770=1196.585,14.580,-44.568,-179.660,5.684,148.903
C04771=1196.580,14.830,-44.582,-179.658,5.685,148.903
C04772=1196.575,15.079,-44.596,-179.656,5.686,148.902
C04773=1196.571,15.328,-44.611,-179.653,5.686,148.901
C04774=1196.566,15.578,-44.626,-179.650,5.687,148.901
C04775=1196.561,15.828,-44.640,-179.648,5.687,148.900
C04776=1196.555,16.077,-44.656,-179.646,5.688,148.899
C04777=1196.550,16.327,-44.670,-179.643,5.688,148.899
C04778=1196.545,16.577,-44.684,-179.640,5.689,148.898
C04779=1196.540,16.826,-44.698,-179.638,5.689,148.897
C04780=1196.536,17.075,-44.713,-179.635,5.690,148.897
C04781=1196.530,17.325,-44.728,-179.633,5.691,148.896
C04782=1196.525,17.575,-44.743,-179.630,5.691,148.896
C04783=1196.521,17.824,-44.758,-179.628,5.692,148.895
C04784=1196.516,18.074,-44.772,-179.625,5.693,148.894
C04785=1196.510,18.322,-44.786,-179.623,5.693,148.894
C04786=1196.505,18.572,-44.801,-179.620,5.694,148.893
C04787=1196.500,18.822,-44.816,-179.617,5.694,148.892
C04788=1196.495,19.071,-44.831,-179.615,5.695,148.892
C04789=1196.490,19.321,-44.845,-179.613,5.696,148.891
C04790=1196.485,19.570,-44.860,-179.610,5.696,148.891
C04791=1196.480,19.820,-44.875,-179.608,5.696,148.890
C04792=1196.475,20.069,-44.890,-179.605,5.696,148.889
C04793=1196.470,20.319,-44.904,-179.603,5.697,148.889
C04794=1196.464,20.569,-44.919,-179.600,5.698,148.888
C04795=1196.460,20.818,-44.934,-179.598,5.698,148.887
C04796=1196.455,21.068,-44.948,-179.595,5.699,148.887
C04797=1196.449,21.317,-44.964,-179.593,5.700,148.886
C04798=1196.445,21.567,-44.978,-179.590,5.700,148.886
C04799=1196.440,21.816,-44.993,-179.588,5.701,148.885
C04800=1196.434,22.066,-45.008,-179.585,5.701,148.884
C04801=1196.430,22.315,-45.023,-179.582,5.702,148.884
C04802=1196.425,22.565,-45.037,-179.580,5.702,148.883
C04803=1196.419,22.814,-45.053,-179.578,5.703,148.882
C04804=1196.414,23.064,-45.067,-179.575,5.703,148.882
C04805=1196.410,23.313,-45.082,-179.572,5.704,148.881
C04806=1196.404,23.562,-45.098,-179.570,5.705,148.881
C04807=1196.400,23.813,-45.112,-179.567,5.705,148.880
C04808=1196.395,24.062,-45.127,-179.565,5.706,148.879
C04809=1196.389,24.312,-45.142,-179.562,5.706,148.879
C04810=1196.385,24.561,-45.157,-179.559,5.708,148.878
C04811=1196.379,24.811,-45.172,-179.557,5.709,148.877
C04812=1196.374,25.060,-45.187,-179.554,5.709,148.877
C04813=1196.370,25.309,-45.202,-179.552,5.710,148.876
C04814=1196.364,25.559,-45.217,-179.549,5.710,148.876
C04815=1196.360,25.808,-45.232,-179.547,5.711,148.875
C04816=1196.354,26.058,-45.247,-179.544,5.711,148.874
C04817=1196.349,26.307,-45.262,-179.541,5.712,148.874
C04818=1196.345,26.556,-45.277,-179.539,5.713,148.873
C04819=1196.339,26.806,-45.292,-179.537,5.713,148.872
C04820=1196.334,27.055,-45.307,-179.534,5.714,148.872
C04821=1196.329,27.306,-45.322,-179.531,5.714,148.871
C04822=1196.325,27.555,-45.337,-179.529,5.715,148.871
C04823=1196.319,27.805,-45.352,-179.527,5.716,148.870
C04824=1196.314,28.054,-45.367,-179.524,5.716,148.869
C04825=1196.309,28.303,-45.383,-179.521,5.717,148.869
C04826=1196.304,28.572,-45.399,-179.519,5.717,148.868
C04827=1196.298,28.841,-45.415,-179.516,5.718,148.867
C04828=1196.293,29.109,-45.431,-179.513,5.718,148.867
C04829=1196.287,29.378,-45.448,-179.510,5.720,148.866
C04830=1196.283,29.627,-45.463,-179.508,5.721,148.865
C04831=1196.277,29.877,-45.478,-179.505,5.721,148.865
C04832=1196.272,30.127,-45.493,-179.503,5.722,148.864
C04833=1196.268,30.377,-45.508,-179.500,5.722,148.863
C04834=1196.263,30.626,-45.523,-179.498,5.723,148.863
C04835=1196.258,30.875,-45.539,-179.495,5.723,148.862
C04836=1196.253,31.124,-45.554,-179.493,5.724,148.862
C04837=1196.247,31.374,-45.569,-179.490,5.724,148.861
C04838=1196.243,31.623,-45.584,-179.488,5.725,148.860
C04839=1196.238,31.873,-45.600,-179.485,5.726,148.860
C04840=1196.232,32.123,-45.615,-179.482,5.726,148.859
C04841=1196.228,32.372,-45.630,-179.480,5.727,148.858
C04842=1196.222,32.621,-45.646,-179.478,5.728,148.858
C04843=1196.218,32.870,-45.661,-179.475,5.728,148.857
C04844=1196.212,33.120,-45.676,-179.472,5.729,148.857
C04845=1196.208,33.370,-45.691,-179.470,5.729,148.856
C04846=1196.203,33.620,-45.707,-179.468,5.730,148.856
C04847=1196.197,33.869,-45.722,-179.465,5.731,148.855
C04848=1196.193,34.118,-45.737,-179.462,5.732,148.854
C04849=1196.187,34.368,-45.753,-179.460,5.733,148.854
C04850=1196.183,34.617,-45.768,-179.457,5.733,148.853
C04851=1196.178,34.867,-45.784,-179.454,5.734,148.852
C04852=1196.172,35.116,-45.800,-179.452,5.735,148.852
C04853=1196.168,35.365,-45.815,-179.449,5.735,148.851
C04854=1196.163,35.615,-45.830,-179.447,5.736,148.851
C04855=1196.157,35.865,-45.846,-179.444,5.736,148.850
C04856=1196.153,36.114,-45.861,-179.442,5.737,148.849
C04857=1196.147,36.363,-45.877,-179.439,5.738,148.849
C04858=1196.143,36.613,-45.893,-179.437,5.738,148.848
C04859=1196.138,36.862,-45.908,-179.434,5.739,148.847
C04860=1196.133,37.112,-45.923,-179.431,5.739,148.847
C04861=1196.127,37.361,-45.939,-179.429,5.740,148.846
C04862=1196.123,37.611,-45.954,-179.426,5.742,148.846
C04863=1196.118,37.860,-45.970,-179.423,5.742,148.845
C04864=1196.112,38.110,-45.985,-179.421,5.743,148.845
C04865=1196.108,38.359,-46.000,-179.419,5.744,148.844
C04866=1196.103,38.609,-46.016,-179.416,5.744,148.843
C04867=1196.098,38.858,-46.032,-179.413,5.745,148.842
C04868=1196.092,39.108,-46.047,-179.411,5.745,148.842
C04869=1196.088,39.357,-46.062,-179.409,5.746,148.841
C04870=1196.083,39.607,-46.078,-179.406,5.747,148.841
C04871=1196.077,39.856,-46.094,-179.404,5.747,148.840
C04872=1196.072,40.106,-46.110,-179.401,5.748,148.840
C04873=1196.068,40.355,-46.126,-179.398,5.749,148.839
C04874=1196.063,40.604,-46.141,-179.395,5.750,148.838
C04875=1196.057,40.854,-46.157,-179.393,5.751,148.838
C04876=1196.053,41.104,-46.173,-179.390,5.751,148.837
C04877=1196.047,41.353,-46.188,-179.388,5.752,148.836
C04878=1196.043,41.602,-46.203,-179.385,5.752,148.836
C04879=1196.038,41.851,-46.220,-179.383,5.753,148.835
C04880=1196.033,42.101,-46.236,-179.380,5.754,148.835
C04881=1196.027,42.351,-46.251,-179.378,5.754,148.834
C04882=1196.022,42.600,-46.267,-179.376,5.755,148.834
C04883=1196.018,42.850,-46.282,-179.372,5.756,148.833
C04884=1196.013,43.099,-46.298,-179.370,5.757,148.832
C04885=1196.008,43.349,-46.314,-179.367,5.757,148.832
C04886=1196.003,43.598,-46.330,-179.365,5.758,148.831
C04887=1195.997,43.848,-46.346,-179.362,5.759,148.830
C04888=1195.993,44.097,-46.362,-179.360,5.759,148.830
C04889=1195.988,44.346,-46.377,-179.358,5.760,148.829
C04890=1195.983,44.596,-46.393,-179.355,5.761,148.829
C04891=1195.978,44.846,-46.409,-179.352,5.761,148.828
C04892=1195.973,45.094,-46.425,-179.349,5.763,148.828
C04893=1195.968,45.344,-46.441,-179.347,5.764,148.827
C04894=1195.963,45.594,-46.457,-179.344,5.764,148.826
C04895=1195.958,45.843,-46.473,-179.342,5.765,148.825
C04896=1195.953,46.093,-46.489,-179.339,5.765,148.825
C04897=1195.948,46.342,-46.504,-179.337,5.766,148.824
C04898=1195.943,46.591,-46.520,-179.334,5.767,148.824
C04899=1195.938,46.841,-46.536,-179.332,5.767,148.823
C04900=1195.933,47.090,-46.552,-179.329,5.769,148.823
C04901=1195.929,47.340,-46.568,-179.326,5.769,148.822
C04902=1195.923,47.589,-46.584,-179.324,5.770,148.821
C04903=1195.918,47.839,-46.600,-179.321,5.771,148.821
C04904=1195.913,48.088,-46.616,-179.319,5.771,148.820
C04905=1195.908,48.337,-46.632,-179.316,5.772,148.819
C04906=1195.903,48.587,-46.648,-179.314,5.773,148.819
C04907=1195.898,48.836,-46.664,-179.311,5.773,148.818
C04908=1195.894,49.086,-46.681,-179.308,5.775,148.818
C04909=1195.888,49.335,-46.696,-179.306,5.775,148.817
C04910=1195.883,49.585,-46.712,-179.303,5.776,148.817
C04911=1195.878,49.834,-46.729,-179.301,5.776,148.816
C04912=1195.873,50.084,-46.745,-179.298,5.777,148.815
C04913=1195.868,50.333,-46.761,-179.296,5.778,148.815
C04914=1195.863,50.582,-46.776,-179.293,5.779,148.814
C04915=1195.859,50.832,-46.793,-179.290,5.780,148.814
C04916=1195.853,51.081,-46.809,-179.288,5.781,148.813
C04917=1195.849,51.331,-46.825,-179.285,5.781,148.812
C04918=1195.843,51.580,-46.841,-179.283,5.782,148.812
C04919=1195.839,51.830,-46.858,-179.280,5.783,148.811
C04920=1195.833,52.079,-46.873,-179.278,5.783,148.811
C04921=1195.829,52.328,-46.890,-179.275,5.784,148.810
C04922=1195.824,52.577,-46.906,-179.272,5.785,148.809
C04923=1195.819,52.827,-46.922,-179.270,5.786,148.809
C04924=1195.814,53.076,-46.938,-179.267,5.786,148.808
C04925=1195.809,53.326,-46.954,-179.265,5.787,148.808
C04926=1195.804,53.575,-46.971,-179.262,5.788,148.807
C04927=1195.799,53.825,-46.987,-179.259,5.789,148.806
C04928=1195.794,54.074,-47.003,-179.257,5.790,148.806
C04929=1195.790,54.323,-47.020,-179.254,5.791,148.805
C04930=1195.783,54.592,-47.037,-179.252,5.791,148.805
C04931=1195.779,54.861,-47.055,-179.249,5.793,148.804
C04932=1195.773,55.129,-47.072,-179.246,5.793,148.803
C04933=1195.768,55.398,-47.089,-179.243,5.794,148.803
C04934=1195.763,55.647,-47.106,-179.241,5.795,148.802
C04935=1195.758,55.896,-47.122,-179.238,5.796,148.802
C04936=1195.753,56.146,-47.139,-179.235,5.796,148.801
C04937=1195.748,56.396,-47.156,-179.233,5.797,148.800
C04938=1195.743,56.645,-47.172,-179.230,5.798,148.800
C04939=1195.739,56.894,-47.189,-179.228,5.798,148.799
C04940=1195.733,57.144,-47.204,-179.225,5.800,148.799
C04941=1195.729,57.393,-47.221,-179.222,5.801,148.798
C04942=1195.723,57.642,-47.238,-179.220,5.801,148.797
C04943=1195.718,57.892,-47.254,-179.218,5.802,148.797
C04944=1195.714,58.142,-47.270,-179.215,5.803,148.796
C04945=1195.709,58.391,-47.287,-179.212,5.803,148.796
C04946=1195.704,58.640,-47.303,-179.210,5.805,148.795
C04947=1195.698,58.889,-47.320,-179.207,5.805,148.794
C04948=1195.693,59.139,-47.336,-179.205,5.806,148.794
C04949=1195.689,59.389,-47.353,-179.202,5.807,148.793
C04950=1195.684,59.637,-47.369,-179.200,5.807,148.793
C04951=1195.679,59.887,-47.386,-179.197,5.809,148.792
C04952=1195.674,60.136,-47.403,-179.194,5.810,148.792
C04953=1195.669,60.386,-47.419,-179.192,5.810,148.791
C04954=1195.664,60.636,-47.435,-179.190,5.811,148.790
C04955=1195.659,60.885,-47.452,-179.187,5.812,148.790
C04956=1195.654,61.134,-47.469,-179.184,5.813,148.789
C04957=1195.650,61.384,-47.486,-179.182,5.814,148.789
C04958=1195.644,61.632,-47.502,-179.179,5.814,148.788
C04959=1195.639,61.882,-47.519,-179.176,5.815,148.787
C04960=1195.634,62.132,-47.535,-179.174,5.817,148.787
C04961=1195.629,62.381,-47.551,-179.171,5.817,148.786
C04962=1195.624,62.631,-47.569,-179.168,5.818,148.786
C04963=1195.620,62.880,-47.585,-179.166,5.819,148.785
C04964=1195.615,63.129,-47.602,-179.163,5.819,148.785
C04965=1195.609,63.379,-47.619,-179.160,5.820,148.784
C04966=1195.605,63.629,-47.636,-179.158,5.821,148.783
C04967=1195.600,63.877,-47.652,-179.155,5.822,148.783
C04968=1195.595,64.127,-47.669,-179.153,5.823,148.782
C04969=1195.590,64.377,-47.686,-179.150,5.824,148.782
C04970=1195.585,64.625,-47.702,-179.147,5.825,148.781
C04971=1195.580,64.875,-47.719,-179.145,5.826,148.781
C04972=1195.575,65.125,-47.736,-179.143,5.826,148.780
C04973=1195.570,65.373,-47.752,-179.140,5.827,148.779
C04974=1195.565,65.623,-47.770,-179.137,5.828,148.779
C04975=1195.561,65.873,-47.786,-179.135,5.829,148.778
C04976=1195.555,66.122,-47.803,-179.132,5.830,148.777
C04977=1195.550,66.371,-47.820,-179.130,5.830,148.777
C04978=1195.546,66.621,-47.836,-179.127,5.832,148.776
C04979=1195.541,66.871,-47.854,-179.125,5.833,148.776
C04980=1195.536,67.120,-47.870,-179.122,5.833,148.775
C04981=1195.530,67.369,-47.887,-179.119,5.834,148.775
C04982=1195.526,67.618,-47.905,-179.117,5.835,148.774
C04983=1195.522,67.867,-47.921,-179.114,5.836,148.774
C04984=1195.516,68.117,-47.939,-179.111,5.837,148.773
C04985=1195.511,68.366,-47.955,-179.109,5.837,148.772
C04986=1195.506,68.616,-47.972,-179.106,5.839,148.772
C04987=1195.502,68.865,-47.989,-179.104,5.840,148.771
C04988=1195.496,69.115,-48.006,-179.101,5.840,148.771
C04989=1195.491,69.364,-48.022,-179.099,5.841,148.770
C04990=1195.486,69.613,-48.040,-179.096,5.843,148.770
C04991=1195.482,69.863,-48.057,-179.093,5.843,148.769
C04992=1195.477,70.112,-48.074,-179.091,5.844,148.768
C04993=1195.472,70.361,-48.091,-179.088,5.845,148.768
C04994=1195.466,70.611,-48.108,-179.085,5.846,148.767
C04995=1195.462,70.860,-48.125,-179.083,5.847,148.767
C04996=1195.457,71.110,-48.143,-179.081,5.847,148.766
C04997=1195.453,71.359,-48.159,-179.078,5.848,148.765
C04998=1195.447,71.608,-48.176,-179.075,5.850,148.765
C04999=1195.443,71.857,-48.194,-179.073,5.850,148.764
C05000=1195.437,72.107,-48.211,-179.070,5.851,148.764
C05001=1195.433,72.356,-48.227,-179.067,5.852,148.763
C05002=1195.428,72.606,-48.245,-179.065,5.853,148.763
C05003=1195.423,72.855,-48.262,-179.062,5.854,148.762
C05004=1195.418,73.104,-48.279,-179.060,5.854,148.762
C05005=1195.412,73.354,-48.296,-179.057,5.856,148.761
C05006=1195.408,73.603,-48.314,-179.054,5.857,148.760
C05007=1195.403,73.853,-48.331,-179.052,5.857,148.760
C05008=1195.399,74.102,-48.348,-179.050,5.858,148.759
C05009=1195.394,74.351,-48.366,-179.046,5.860,148.759
C05010=1195.388,74.601,-48.383,-179.044,5.860,148.758
C05011=1195.383,74.850,-48.399,-179.042,5.861,148.758
C05012=1195.378,75.099,-48.417,-179.038,5.862,148.757
C05013=1195.374,75.348,-48.434,-179.036,5.863,148.757
C05014=1195.369,75.598,-48.451,-179.034,5.864,148.756
C05015=1195.364,75.847,-48.469,-179.031,5.866,148.755
C05016=1195.359,76.097,-48.486,-179.028,5.866,148.755
C05017=1195.354,76.346,-48.504,-179.026,5.867,148.754
C05018=1195.349,76.596,-48.521,-179.024,5.868,148.754
C05019=1195.344,76.844,-48.538,-179.020,5.869,148.753
C05020=1195.339,77.094,-48.555,-179.018,5.870,148.753
C05021=1195.334,77.344,-48.572,-179.016,5.870,148.752
C05022=1195.330,77.592,-48.590,-179.012,5.872,148.751
C05023=1195.325,77.842,-48.607,-179.010,5.873,148.751
C05024=1195.320,78.091,-48.625,-179.008,5.873,148.750
C05025=1195.315,78.341,-48.642,-179.005,5.875,148.750
C05026=1195.310,78.590,-48.660,-179.002,5.876,148.749
C05027=1195.305,78.840,-48.677,-179.000,5.876,148.749
C05028=1195.300,79.089,-48.695,-178.998,5.877,148.748
C05029=1195.296,79.339,-48.712,-178.994,5.878,148.747
C05030=1195.291,79.588,-48.730,-178.992,5.879,148.747
C05031=1195.286,79.838,-48.747,-178.990,5.880,148.746
C05032=1195.280,80.086,-48.765,-178.987,5.882,148.746
C05033=1195.276,80.335,-48.782,-178.984,5.882,148.745
C05034=1195.271,80.604,-48.801,-178.981,5.883,148.745
C05035=1195.265,80.872,-48.820,-178.979,5.884,148.744
C05036=1195.260,81.141,-48.839,-178.976,5.886,148.744
C05037=1195.255,81.410,-48.857,-178.973,5.886,148.743
C05038=1195.250,81.659,-48.875,-178.970,5.887,148.742
C05039=1195.246,81.908,-48.893,-178.968,5.889,148.742
C05040=1195.240,82.158,-48.910,-178.965,5.889,148.741
C05041=1195.235,82.407,-48.928,-178.963,5.890,148.741
C05042=1195.231,82.656,-48.946,-178.960,5.891,148.740
C05043=1195.225,82.906,-48.963,-178.958,5.892,148.740
C05044=1195.220,83.155,-48.981,-178.955,5.893,148.739
C05045=1195.216,83.404,-48.999,-178.952,5.895,148.739
C05046=1195.211,83.654,-49.016,-178.950,5.895,148.738
C05047=1195.206,83.903,-49.034,-178.947,5.896,148.737
C05048=1195.201,84.152,-49.052,-178.944,5.897,148.737
C05049=1195.196,84.402,-49.069,-178.942,5.898,148.736
C05050=1195.191,84.651,-49.087,-178.940,5.899,148.736
C05051=1195.186,84.900,-49.105,-178.936,5.900,148.735
C05052=1195.182,85.149,-49.122,-178.934,5.901,148.735
C05053=1195.177,85.399,-49.140,-178.932,5.902,148.734
C05054=1195.172,85.648,-49.158,-178.929,5.904,148.734
C05055=1195.167,85.897,-49.176,-178.926,5.904,148.733
C05056=1195.162,86.146,-49.194,-178.924,5.905,148.732
C05057=1195.157,86.395,-49.212,-178.921,5.906,148.732
C05058=1195.152,86.645,-49.229,-178.918,5.907,148.731
C05059=1195.147,86.894,-49.247,-178.916,5.909,148.731
C05060=1195.142,87.144,-49.265,-178.913,5.909,148.730
C05061=1195.137,87.393,-49.283,-178.911,5.910,148.730
C05062=1195.132,87.642,-49.301,-178.908,5.912,148.729
C05063=1195.127,87.892,-49.318,-178.905,5.912,148.729
C05064=1195.122,88.141,-49.336,-178.903,5.913,148.728
C05065=1195.119,88.390,-49.354,-178.900,5.915,148.728
C05066=1195.114,88.640,-49.372,-178.898,5.915,148.727
C05067=1195.109,88.889,-49.390,-178.895,5.916,148.727
C05068=1195.104,89.138,-49.408,-178.892,5.918,148.726
C05069=1195.099,89.387,-49.426,-178.890,5.918,148.725
C05070=1195.094,89.636,-49.444,-178.887,5.920,148.725
C05071=1195.089,89.885,-49.462,-178.884,5.920,148.724
C05072=1195.084,90.135,-49.480,-178.882,5.921,148.724
C05073=1195.079,90.384,-49.497,-178.879,5.923,148.723
C05074=1195.075,90.634,-49.515,-178.877,5.924,148.723
C05075=1195.070,90.884,-49.533,-178.874,5.924,148.722
C05076=1195.064,91.133,-49.552,-178.871,5.926,148.722
C05077=1195.059,91.382,-49.570,-178.869,5.927,148.721
C05078=1195.054,91.631,-49.588,-178.866,5.928,148.721
C05079=1195.049,91.881,-49.606,-178.863,5.929,148.720
C05080=1195.044,92.130,-49.624,-178.861,5.930,148.720
C05081=1195.040,92.380,-49.642,-178.858,5.931,148.719
C05082=1195.035,92.629,-49.660,-178.856,5.932,148.718
C05083=1195.030,92.878,-49.678,-178.853,5.933,148.718
C05084=1195.025,93.127,-49.696,-178.851,5.934,148.717
C05085=1195.020,93.376,-49.714,-178.848,5.935,148.717
C05086=1195.016,93.625,-49.733,-178.845,5.937,148.716
C05087=1195.012,93.875,-49.751,-178.843,5.937,148.716
C05088=1195.007,94.124,-49.769,-178.840,5.939,148.715
C05089=1195.001,94.373,-49.788,-178.837,5.940,148.715
C05090=1194.996,94.623,-49.806,-178.835,5.940,148.714
C05091=1194.991,94.872,-49.824,-178.832,5.942,148.714
C05092=1194.987,95.122,-49.842,-178.830,5.943,148.713
C05093=1194.982,95.371,-49.860,-178.827,5.944,148.712
C05094=1194.977,95.620,-49.878,-178.825,5.945,148.712
C05095=1194.972,95.869,-49.897,-178.822,5.946,148.711
C05096=1194.967,96.118,-49.915,-178.819,5.947,148.711
C05097=1194.962,96.368,-49.933,-178.817,5.948,148.710
C05098=1194.958,96.617,-49.951,-178.814,5.950,148.710
C05099=1194.953,96.866,-49.969,-178.811,5.950,148.709
C05100=1194.948,97.115,-49.987,-178.809,5.952,148.709
C05101=1194.943,97.365,-50.007,-178.806,5.953,148.708
C05102=1194.938,97.614,-50.025,-178.804,5.953,148.708
C05103=1194.933,97.863,-50.043,-178.801,5.955,148.707
C05104=1194.928,98.113,-50.061,-178.799,5.956,148.707
C05105=1194.924,98.362,-50.080,-178.795,5.957,148.706
C05106=1194.919,98.611,-50.099,-178.793,5.958,148.706
C05107=1194.914,98.860,-50.117,-178.790,5.959,148.705
C05108=1194.909,99.110,-50.135,-178.788,5.960,148.705
C05109=1194.905,99.359,-50.154,-178.785,5.961,148.704
C05110=1194.899,99.608,-50.172,-178.783,5.963,148.704
C05111=1194.894,99.858,-50.190,-178.780,5.963,148.703
C05112=1194.890,100.106,-50.209,-178.777,5.965,148.703
C05113=1194.885,100.356,-50.228,-178.775,5.966,148.702
C05114=1194.880,100.605,-50.246,-178.772,5.967,148.701
C05115=1194.875,100.854,-50.265,-178.769,5.968,148.701
C05116=1194.871,101.104,-50.283,-178.767,5.969,148.700
C05117=1194.865,101.353,-50.301,-178.764,5.970,148.700
C05118=1194.860,101.602,-50.320,-178.762,5.971,148.699
C05119=1194.856,101.852,-50.339,-178.759,5.973,148.699
C05120=1194.850,102.101,-50.357,-178.757,5.973,148.698
C05121=1194.846,102.350,-50.376,-178.753,5.975,148.698
C05122=1194.842,102.600,-50.394,-178.751,5.976,148.697
C05123=1194.836,102.849,-50.413,-178.749,5.978,148.697
C05124=1194.831,103.098,-50.431,-178.746,5.978,148.696
C05125=1194.827,103.347,-50.450,-178.743,5.980,148.696
C05126=1194.822,103.597,-50.469,-178.741,5.980,148.695
C05127=1194.817,103.846,-50.487,-178.738,5.981,148.695
C05128=1194.812,104.095,-50.507,-178.735,5.983,148.694
C05129=1194.807,104.344,-50.525,-178.733,5.984,148.694
C05130=1194.802,104.593,-50.543,-178.730,5.985,148.693
C05131=1194.797,104.843,-50.562,-178.728,5.986,148.693
C05132=1194.793,105.092,-50.581,-178.725,5.987,148.692
C05133=1194.788,105.342,-50.600,-178.723,5.988,148.692
C05134=1194.783,105.590,-50.619,-178.720,5.990,148.691
C05135=1194.778,105.840,-50.637,-178.717,5.991,148.691
C05136=1194.774,106.089,-50.656,-178.714,5.992,148.690
C05137=1194.769,106.338,-50.675,-178.712,5.993,148.689
C05138=1194.763,106.606,-50.695,-178.709,5.995,148.689
C05139=1194.758,106.876,-50.715,-178.707,5.995,148.688
C05140=1194.753,107.143,-50.735,-178.703,5.997,148.688
C05141=1194.748,107.413,-50.756,-178.701,5.998,148.687
C05142=1194.743,107.661,-50.775,-178.698,5.999,148.687
C05143=1194.738,107.910,-50.794,-178.695,6.001,148.686
C05144=1194.734,108.160,-50.812,-178.693,6.001,148.686
C05145=1194.728,108.409,-50.831,-178.690,6.003,148.685
C05146=1194.724,108.658,-50.851,-178.687,6.004,148.685
C05147=1194.719,108.907,-50.869,-178.685,6.005,148.684
C05148=1194.715,109.157,-50.888,-178.683,6.006,148.684
C05149=1194.709,109.406,-50.907,-178.679,6.008,148.683
C05150=1194.704,109.655,-50.925,-178.677,6.009,148.683
C05151=1194.700,109.904,-50.945,-178.674,6.010,148.682
C05152=1194.695,110.153,-50.964,-178.672,6.011,148.682
C05153=1194.690,110.403,-50.983,-178.669,6.012,148.681
C05154=1194.685,110.652,-51.002,-178.667,6.013,148.681
C05155=1194.681,110.901,-51.021,-178.664,6.015,148.680
C05156=1194.675,111.150,-51.040,-178.661,6.016,148.680
C05157=1194.671,111.400,-51.059,-178.659,6.017,148.679
C05158=1194.666,111.649,-51.078,-178.656,6.018,148.679
C05159=1194.662,111.898,-51.097,-178.653,6.020,148.678
C05160=1194.656,112.147,-51.116,-178.651,6.020,148.678
C05161=1194.651,112.397,-51.135,-178.648,6.022,148.677
C05162=1194.647,112.646,-51.154,-178.646,6.023,148.677
C05163=1194.642,112.895,-51.174,-178.643,6.024,148.676
C05164=1194.637,113.144,-51.193,-178.641,6.025,148.676
C05165=1194.633,113.393,-51.212,-178.637,6.027,148.675
C05166=1194.627,113.643,-51.231,-178.635,6.028,148.675
C05167=1194.623,113.892,-51.250,-178.633,6.029,148.674
C05168=1194.618,114.141,-51.269,-178.630,6.030,148.674
C05169=1194.613,114.391,-51.289,-178.627,6.032,148.673
C05170=1194.608,114.639,-51.307,-178.624,6.033,148.673
C05171=1194.603,114.889,-51.327,-178.622,6.034,148.672
C05172=1194.598,115.137,-51.346,-178.619,6.036,148.672
C05173=1194.594,115.387,-51.365,-178.617,6.036,148.671
C05174=1194.589,115.636,-51.385,-178.614,6.038,148.671
C05175=1194.584,115.886,-51.403,-178.611,6.039,148.670
C05176=1194.579,116.135,-51.423,-178.609,6.041,148.670
C05177=1194.574,116.384,-51.442,-178.606,6.041,148.669
C05178=1194.570,116.634,-51.462,-178.603,6.043,148.669
C05179=1194.564,116.882,-51.481,-178.601,6.044,148.668
C05180=1194.560,117.132,-51.500,-178.598,6.045,148.668
C05181=1194.555,117.381,-51.520,-178.596,6.046,148.667
C05182=1194.550,117.630,-51.539,-178.593,6.048,148.667
C05183=1194.545,117.880,-51.558,-178.590,6.049,148.666
C05184=1194.541,118.128,-51.577,-178.588,6.050,148.666
C05185=1194.536,118.378,-51.597,-178.585,6.052,148.665
C05186=1194.531,118.627,-51.616,-178.583,6.053,148.665
C05187=1194.526,118.876,-51.636,-178.580,6.054,148.664
C05188=1194.521,119.126,-51.655,-178.577,6.055,148.664
C05189=1194.517,119.374,-51.674,-178.575,6.057,148.663
C05190=1194.512,119.623,-51.694,-178.572,6.058,148.663
C05191=1194.507,119.873,-51.714,-178.569,6.059,148.662
C05192=1194.502,120.122,-51.733,-178.567,6.061,148.662
C05193=1194.497,120.371,-51.753,-178.564,6.062,148.662
C05194=1194.493,120.621,-51.772,-178.561,6.063,148.661
C05195=1194.488,120.869,-51.791,-178.559,6.064,148.660
C05196=1194.483,121.119,-51.811,-178.556,6.065,148.660
C05197=1194.479,121.369,-51.831,-178.554,6.066,148.659
C05198=1194.473,121.617,-51.851,-178.551,6.068,148.659
C05199=1194.469,121.866,-51.870,-178.548,6.070,148.658
C05200=1194.464,122.116,-51.890,-178.546,6.070,148.658
C05201=1194.459,122.364,-51.909,-178.543,6.072,148.658
C05202=1194.455,122.614,-51.928,-178.540,6.073,148.657
C05203=1194.450,122.864,-51.948,-178.538,6.075,148.657
C05204=1194.445,123.112,-51.968,-178.536,6.076,148.656
C05205=1194.440,123.361,-51.988,-178.532,6.077,148.656
C05206=1194.435,123.611,-52.007,-178.530,6.079,148.655
C05207=1194.430,123.860,-52.027,-178.527,6.079,148.655
C05208=1194.426,124.109,-52.047,-178.525,6.081,148.654
C05209=1194.421,124.358,-52.067,-178.522,6.082,148.654
C05210=1194.416,124.607,-52.086,-178.519,6.083,148.653
C05211=1194.411,124.857,-52.106,-178.517,6.085,148.653
C05212=1194.407,125.105,-52.125,-178.514,6.086,148.652
C05213=1194.402,125.355,-52.145,-178.511,6.087,148.652
C05214=1194.397,125.604,-52.164,-178.509,6.088,148.651
C05215=1194.393,125.853,-52.185,-178.506,6.090,148.651
C05216=1194.388,126.102,-52.204,-178.503,6.092,148.650
C05217=1194.383,126.352,-52.224,-178.501,6.093,148.650
C05218=1194.378,126.600,-52.244,-178.498,6.094,148.649
C05219=1194.373,126.850,-52.264,-178.496,6.095,148.649
C05220=1194.369,127.099,-52.284,-178.493,6.097,148.648
C05221=1194.364,127.348,-52.304,-178.490,6.098,148.648
C05222=1194.359,127.597,-52.323,-178.488,6.099,148.647
C05223=1194.354,127.846,-52.343,-178.485,6.101,148.647
C05224=1194.350,128.096,-52.363,-178.483,6.102,148.647
C05225=1194.345,128.345,-52.383,-178.480,6.103,148.646
C05226=1194.340,128.594,-52.403,-178.477,6.105,148.646
C05227=1194.335,128.843,-52.422,-178.475,6.106,148.645
C05228=1194.330,129.092,-52.443,-178.472,6.107,148.645
C05229=1194.325,129.342,-52.463,-178.469,6.109,148.644
C05230=1194.321,129.591,-52.483,-178.467,6.110,148.644
C05231=1194.316,129.840,-52.503,-178.464,6.111,148.643
C05232=1194.311,130.089,-52.523,-178.462,6.112,148.643
C05233=1194.306,130.338,-52.543,-178.459,6.114,148.642
C05234=1194.302,130.587,-52.563,-178.456,6.116,148.642
C05235=1194.297,130.837,-52.583,-178.454,6.116,148.641
C05236=1194.293,131.086,-52.603,-178.451,6.118,148.641
C05237=1194.287,131.335,-52.622,-178.448,6.120,148.641
C05238=1194.282,131.584,-52.643,-178.446,6.121,148.640
C05239=1194.278,131.833,-52.664,-178.443,6.122,148.640
C05240=1194.273,132.082,-52.683,-178.440,6.124,148.639
C05241=1194.268,132.331,-52.704,-178.438,6.125,148.639
C05242=1194.263,132.600,-52.725,-178.435,6.126,148.638
C05243=1194.258,132.868,-52.747,-178.432,6.128,148.638
C05244=1194.253,133.137,-52.769,-178.429,6.130,148.637
C05245=1194.248,133.406,-52.790,-178.426,6.131,148.637
C05246=1194.243,133.655,-52.810,-178.424,6.132,148.636
C05247=1194.238,133.904,-52.831,-178.421,6.134,148.636
C05248=1194.233,134.154,-52.851,-178.419,6.136,148.635
C05249=1194.229,134.403,-52.871,-178.416,6.136,148.635
C05250=1194.224,134.651,-52.891,-178.413,6.138,148.634
C05251=1194.219,134.900,-52.911,-178.411,6.140,148.634
C05252=1194.214,135.150,-52.932,-178.408,6.140,148.633
C05253=1194.209,135.399,-52.952,-178.405,6.142,148.633
C05254=1194.205,135.648,-52.973,-178.403,6.144,148.633
C05255=1194.200,135.897,-52.992,-178.400,6.145,148.632
C05256=1194.195,136.146,-53.013,-178.397,6.146,148.632
C05257=1194.191,136.395,-53.034,-178.395,6.148,148.631
C05258=1194.186,136.644,-53.054,-178.392,6.149,148.631
C05259=1194.181,136.894,-53.074,-178.389,6.150,148.630
C05260=1194.176,137.143,-53.095,-178.387,6.152,148.630
C05261=1194.172,137.392,-53.115,-178.384,6.153,148.629
C05262=1194.167,137.640,-53.135,-178.382,6.155,148.629
C05263=1194.162,137.890,-53.156,-178.379,6.156,148.628
C05264=1194.157,138.139,-53.176,-178.377,6.157,148.628
C05265=1194.152,138.388,-53.196,-178.374,6.159,148.628
C05266=1194.147,138.637,-53.217,-178.371,6.161,148.627
C05267=1194.143,138.886,-53.237,-178.369,6.161,148.627
C05268=1194.138,139.135,-53.258,-178.366,6.163,148.626
C05269=1194.133,139.385,-53.279,-178.363,6.165,148.626
C05270=1194.129,139.633,-53.299,-178.361,6.166,148.625
C05271=1194.124,139.883,-53.319,-178.358,6.167,148.625
C05272=1194.119,140.132,-53.340,-178.355,6.169,148.624
C05273=1194.114,140.381,-53.360,-178.353,6.170,148.624
C05274=1194.110,140.630,-53.381,-178.350,6.172,148.624
C05275=1194.105,140.879,-53.401,-178.347,6.173,148.623
C05276=1194.100,141.128,-53.422,-178.345,6.175,148.623
C05277=1194.095,141.378,-53.443,-178.342,6.176,148.622
C05278=1194.091,141.627,-53.463,-178.340,6.178,148.622
C05279=1194.086,141.876,-53.484,-178.337,6.179,148.621
C05280=1194.081,142.125,-53.505,-178.334,6.180,148.621
C05281=1194.077,142.374,-53.525,-178.332,6.182,148.620
C05282=1194.072,142.623,-53.546,-178.329,6.184,148.620
C05283=1194.067,142.872,-53.566,-178.326,6.184,148.619
C05284=1194.062,143.121,-53.587,-178.324,6.186,148.619
C05285=1194.057,143.370,-53.608,-178.321,6.188,148.619
C05286=1194.053,143.619,-53.628,-178.318,6.189,148.618
C05287=1194.048,143.869,-53.649,-178.316,6.190,148.618
C05288=1194.044,144.118,-53.670,-178.313,6.192,148.617
C05289=1194.039,144.367,-53.691,-178.310,6.194,148.617
C05290=1194.034,144.616,-53.711,-178.308,6.195,148.617
C05291=1194.030,144.865,-53.733,-178.305,6.196,148.616
C05292=1194.025,145.114,-53.753,-178.302,6.198,148.616
C05293=1194.020,145.363,-53.774,-178.300,6.200,148.615
C05294=1194.016,145.612,-53.794,-178.298,6.200,148.615
C05295=1194.010,145.861,-53.815,-178.295,6.202,148.614
C05296=1194.006,146.110,-53.836,-178.292,6.204,148.614
C05297=1194.001,146.360,-53.857,-178.289,6.205,148.613
C05298=1193.996,146.608,-53.878,-178.287,6.206,148.613
C05299=1193.992,146.858,-53.899,-178.284,6.208,148.613
C05300=1193.987,147.107,-53.920,-178.282,6.210,148.612
C05301=1193.982,147.356,-53.940,-178.278,6.211,148.612
C05302=1193.977,147.605,-53.961,-178.276,6.212,148.611
C05303=1193.973,147.854,-53.983,-178.274,6.214,148.611
C05304=1193.968,148.103,-54.003,-178.271,6.216,148.610
C05305=1193.963,148.352,-54.024,-178.268,6.218,148.610
C05306=1193.958,148.601,-54.045,-178.266,6.218,148.609
C05307=1193.954,148.850,-54.067,-178.263,6.220,148.609
C05308=1193.950,149.099,-54.087,-178.260,6.222,148.609
C05309=1193.944,149.349,-54.108,-178.258,6.224,148.608
C05310=1193.939,149.598,-54.129,-178.256,6.225,148.608
C05311=1193.935,149.846,-54.150,-178.252,6.226,148.607
C05312=1193.930,150.095,-54.171,-178.250,6.228,148.607
C05313=1193.925,150.345,-54.193,-178.247,6.230,148.607
C05314=1193.921,150.594,-54.214,-178.245,6.230,148.606
C05315=1193.916,150.843,-54.235,-178.242,6.232,148.606
C05316=1193.911,151.092,-54.256,-178.239,6.234,148.605
C05317=1193.907,151.341,-54.277,-178.236,6.235,148.605
C05318=1193.902,151.590,-54.298,-178.234,6.236,148.604
C05319=1193.897,151.839,-54.320,-178.232,6.238,148.604
C05320=1193.893,152.088,-54.340,-178.229,6.240,148.604
C05321=1193.888,152.337,-54.361,-178.226,6.241,148.603
C05322=1193.883,152.586,-54.383,-178.223,6.243,148.603
C05323=1193.878,152.835,-54.404,-178.221,6.244,148.602
C05324=1193.874,153.084,-54.425,-178.218,6.246,148.602
C05325=1193.869,153.334,-54.446,-178.216,6.248,148.602
C05326=1193.864,153.582,-54.468,-178.213,6.249,148.601
C05327=1193.859,153.832,-54.489,-178.210,6.250,148.601
C05328=1193.855,154.081,-54.510,-178.208,6.252,148.600
C05329=1193.850,154.330,-54.531,-178.205,6.254,148.600
C05330=1193.845,154.578,-54.553,-178.202,6.255,148.599
C05331=1193.840,154.828,-54.574,-178.200,6.257,148.599
C05332=1193.836,155.077,-54.596,-178.198,6.258,148.599
C05333=1193.831,155.326,-54.616,-178.194,6.260,148.598
C05334=1193.827,155.575,-54.638,-178.192,6.261,148.598
C05335=1193.821,155.824,-54.659,-178.189,6.263,148.597
C05336=1193.817,156.073,-54.681,-178.186,6.265,148.597
C05337=1193.812,156.322,-54.703,-178.184,6.266,148.597
C05338=1193.808,156.571,-54.723,-178.182,6.268,148.596
C05339=1193.804,156.820,-54.745,-178.179,6.269,148.596
C05340=1193.798,157.069,-54.766,-178.176,6.271,148.595
C05341=1193.794,157.318,-54.788,-178.173,6.273,148.595
C05342=1193.789,157.567,-54.809,-178.171,6.274,148.594
C05343=1193.784,157.817,-54.831,-178.168,6.275,148.594
C05344=1193.779,158.065,-54.852,-178.166,6.277,148.594
C05345=1193.774,158.314,-54.874,-178.163,6.279,148.593
C05346=1193.770,158.583,-54.897,-178.160,6.280,148.593
C05347=1193.764,158.852,-54.920,-178.157,6.282,148.592
C05348=1193.759,159.121,-54.943,-178.154,6.284,148.592
C05349=1193.754,159.390,-54.967,-178.151,6.285,148.591
C05350=1193.749,159.639,-54.988,-178.149,6.287,148.591
C05351=1193.745,159.888,-55.009,-178.146,6.289,148.591
C05352=1193.741,160.137,-55.031,-178.144,6.290,148.590
C05353=1193.736,160.386,-55.053,-178.141,6.292,148.590
C05354=1193.731,160.636,-55.074,-178.138,6.294,148.590
C05355=1193.726,160.884,-55.096,-178.136,6.295,148.589
C05356=1193.722,161.134,-55.118,-178.133,6.297,148.589
C05357=1193.717,161.382,-55.140,-178.130,6.299,148.588
C05358=1193.712,161.631,-55.161,-178.128,6.300,148.588
C05359=1193.708,161.881,-55.183,-178.125,6.301,148.587
C05360=1193.703,162.130,-55.204,-178.122,6.303,148.587
C05361=1193.699,162.379,-55.226,-178.120,6.305,148.587
C05362=1193.694,162.628,-55.248,-178.117,6.307,148.586
C05363=1193.689,162.876,-55.270,-178.114,6.308,148.586
C05364=1193.685,163.126,-55.292,-178.112,6.310,148.586
C05365=1193.680,163.374,-55.313,-178.110,6.311,148.585
C05366=1193.675,163.623,-55.335,-178.106,6.313,148.585
C05367=1193.670,163.873,-55.356,-178.104,6.314,148.584
C05368=1193.665,164.121,-55.378,-178.101,6.316,148.584
C05369=1193.661,164.371,-55.400,-178.098,6.318,148.583
C05370=1193.656,164.619,-55.422,-178.096,6.320,148.583
C05371=1193.652,164.869,-55.444,-178.094,6.321,148.583
C05372=1193.646,165.118,-55.466,-178.091,6.323,148.582
C05373=1193.642,165.367,-55.488,-178.088,6.324,148.582
C05374=1193.637,165.616,-55.510,-178.086,6.326,148.582
C05375=1193.633,165.865,-55.532,-178.083,6.328,148.581
C05376=1193.628,166.114,-55.554,-178.080,6.329,148.581
C05377=1193.623,166.362,-55.575,-178.077,6.331,148.580
C05378=1193.619,166.612,-55.597,-178.074,6.333,148.580
C05379=1193.614,166.860,-55.619,-178.072,6.334,148.580
C05380=1193.610,167.110,-55.641,-178.070,6.336,148.579
C05381=1193.604,167.359,-55.663,-178.067,6.337,148.579
C05382=1193.600,167.608,-55.685,-178.064,6.339,148.578
C05383=1193.595,167.857,-55.707,-178.062,6.341,148.578
C05384=1193.591,168.106,-55.729,-178.059,6.343,148.578
C05385=1193.586,168.354,-55.752,-178.056,6.345,148.577
C05386=1193.582,168.603,-55.774,-178.054,6.346,148.577
C05387=1193.576,168.852,-55.796,-178.051,6.347,148.577
C05388=1193.572,169.102,-55.818,-178.049,6.349,148.576
C05389=1193.567,169.350,-55.840,-178.046,6.351,148.576
C05390=1193.563,169.600,-55.862,-178.043,6.352,148.575
C05391=1193.558,169.848,-55.883,-178.040,6.354,148.575
C05392=1193.553,170.097,-55.907,-178.038,6.356,148.575
C05393=1193.549,170.346,-55.928,-178.035,6.358,148.574
C05394=1193.544,170.595,-55.950,-178.032,6.360,148.574
C05395=1193.540,170.844,-55.972,-178.030,6.361,148.573
C05396=1193.534,171.093,-55.995,-178.028,6.362,148.573
C05397=1193.530,171.342,-56.017,-178.025,6.364,148.573
C05398=1193.526,171.591,-56.039,-178.022,6.366,148.572
C05399=1193.521,171.840,-56.062,-178.020,6.368,148.572
C05400=1193.516,172.089,-56.084,-178.017,6.369,148.572
C05401=1193.512,172.338,-56.106,-178.014,6.371,148.571
C05402=1193.507,172.586,-56.128,-178.012,6.373,148.571
C05403=1193.502,172.836,-56.151,-178.009,6.375,148.570
C05404=1193.498,173.085,-56.173,-178.006,6.377,148.570
C05405=1193.493,173.333,-56.195,-178.003,6.378,148.570
C05406=1193.488,173.583,-56.218,-178.001,6.380,148.569
C05407=1193.483,173.832,-56.239,-177.999,6.381,148.569
C05408=1193.479,174.080,-56.262,-177.996,6.383,148.569
C05409=1193.474,174.330,-56.285,-177.993,6.384,148.568
C05410=1193.470,174.578,-56.307,-177.990,6.386,148.568
C05411=1193.465,174.827,-56.329,-177.988,6.388,148.567
C05412=1193.460,175.076,-56.351,-177.985,6.390,148.567
C05413=1193.456,175.325,-56.374,-177.982,6.392,148.567
C05414=1193.451,175.575,-56.397,-177.980,6.393,148.566
C05415=1193.446,175.823,-56.419,-177.977,6.395,148.566
C05416=1193.442,176.072,-56.441,-177.974,6.397,148.566
C05417=1193.437,176.322,-56.464,-177.972,6.399,148.565
C05418=1193.432,176.570,-56.486,-177.969,6.401,148.565
C05419=1193.427,176.820,-56.509,-177.966,6.402,148.564
C05420=1193.423,177.068,-56.532,-177.964,6.404,148.564
C05421=1193.418,177.317,-56.554,-177.961,6.406,148.564
C05422=1193.414,177.566,-56.577,-177.959,6.407,148.563
C05423=1193.410,177.815,-56.599,-177.956,6.409,148.563
C05424=1193.404,178.064,-56.622,-177.953,6.410,148.563
C05425=1193.400,178.313,-56.644,-177.951,6.412,148.562
C05426=1193.395,178.562,-56.667,-177.948,6.414,148.562
C05427=1193.390,178.811,-56.689,-177.945,6.416,148.562
C05428=1193.386,179.060,-56.712,-177.943,6.418,148.561
C05429=1193.382,179.308,-56.735,-177.940,6.419,148.561
C05430=1193.376,179.557,-56.757,-177.937,6.421,148.560
C05431=1193.372,179.806,-56.780,-177.935,6.423,148.560
C05432=1193.367,180.056,-56.803,-177.932,6.425,148.560
C05433=1193.363,180.304,-56.826,-177.929,6.427,148.559
C05434=1193.358,180.553,-56.849,-177.927,6.428,148.559
C05435=1193.354,180.802,-56.871,-177.924,6.430,148.559
C05436=1193.349,181.051,-56.894,-177.921,6.432,148.558
C05437=1193.345,181.300,-56.917,-177.919,6.434,148.558
C05438=1193.339,181.549,-56.939,-177.916,6.436,148.558
C05439=1193.335,181.798,-56.962,-177.913,6.437,148.557
C05440=1193.331,182.047,-56.985,-177.911,6.439,148.557
C05441=1193.326,182.296,-57.008,-177.908,6.441,148.557
C05442=1193.321,182.544,-57.030,-177.905,6.443,148.556
C05443=1193.316,182.793,-57.054,-177.903,6.445,148.556
C05444=1193.312,183.042,-57.077,-177.900,6.446,148.555
C05445=1193.307,183.292,-57.099,-177.897,6.448,148.555
C05446=1193.302,183.540,-57.122,-177.895,6.450,148.555
C05447=1193.298,183.789,-57.145,-177.892,6.452,148.554
C05448=1193.294,184.038,-57.168,-177.890,6.454,148.554
C05449=1193.289,184.287,-57.191,-177.887,6.456,148.554
C05450=1193.284,184.556,-57.216,-177.884,6.457,148.553
C05451=1193.279,184.826,-57.241,-177.881,6.459,148.553
C05452=1193.274,185.095,-57.265,-177.879,6.461,148.553
C05453=1193.269,185.365,-57.290,-177.876,6.463,148.552
C05454=1193.264,185.614,-57.314,-177.873,6.465,148.552
C05455=1193.260,185.863,-57.336,-177.870,6.467,148.552
C05456=1193.255,186.112,-57.359,-177.868,6.469,148.551
C05457=1193.250,186.361,-57.382,-177.865,6.471,148.551
C05458=1193.245,186.610,-57.405,-177.862,6.472,148.551
C05459=1193.241,186.859,-57.428,-177.860,6.474,148.550
C05460=1193.237,187.108,-57.452,-177.857,6.476,148.550
C05461=1193.232,187.357,-57.475,-177.854,6.478,148.549
C05462=1193.227,187.605,-57.498,-177.852,6.480,148.549
C05463=1193.223,187.854,-57.521,-177.849,6.482,148.549
C05464=1193.218,188.103,-57.544,-177.847,6.484,148.549
C05465=1193.213,188.352,-57.567,-177.844,6.485,148.548
C05466=1193.209,188.601,-57.591,-177.841,6.487,148.548
C05467=1193.205,188.850,-57.614,-177.839,6.489,148.548
C05468=1193.200,189.099,-57.637,-177.836,6.491,148.547
C05469=1193.195,189.348,-57.660,-177.833,6.493,148.547
C05470=1193.190,189.596,-57.683,-177.831,6.494,148.547
C05471=1193.185,189.845,-57.707,-177.828,6.496,148.546
C05472=1193.181,190.094,-57.729,-177.825,6.498,148.546
C05473=1193.177,190.343,-57.753,-177.823,6.500,148.545
C05474=1193.172,190.592,-57.776,-177.820,6.502,148.545
C05475=1193.167,190.841,-57.799,-177.817,6.503,148.545
C05476=1193.163,191.090,-57.823,-177.815,6.506,148.545
C05477=1193.158,191.339,-57.846,-177.813,6.507,148.544
C05478=1193.153,191.588,-57.870,-177.810,6.509,148.544
C05479=1193.149,191.836,-57.893,-177.807,6.511,148.544
C05480=1193.145,192.085,-57.916,-177.805,6.513,148.543
C05481=1193.139,192.333,-57.939,-177.802,6.515,148.543
C05482=1193.135,192.582,-57.963,-177.799,6.516,148.543
C05483=1193.130,192.831,-57.986,-177.797,6.518,148.542
C05484=1193.125,193.080,-58.009,-177.794,6.520,148.542
C05485=1193.121,193.329,-58.034,-177.791,6.522,148.541
C05486=1193.116,193.578,-58.057,-177.789,6.524,148.541
C05487=1193.112,193.827,-58.080,-177.786,6.526,148.541
